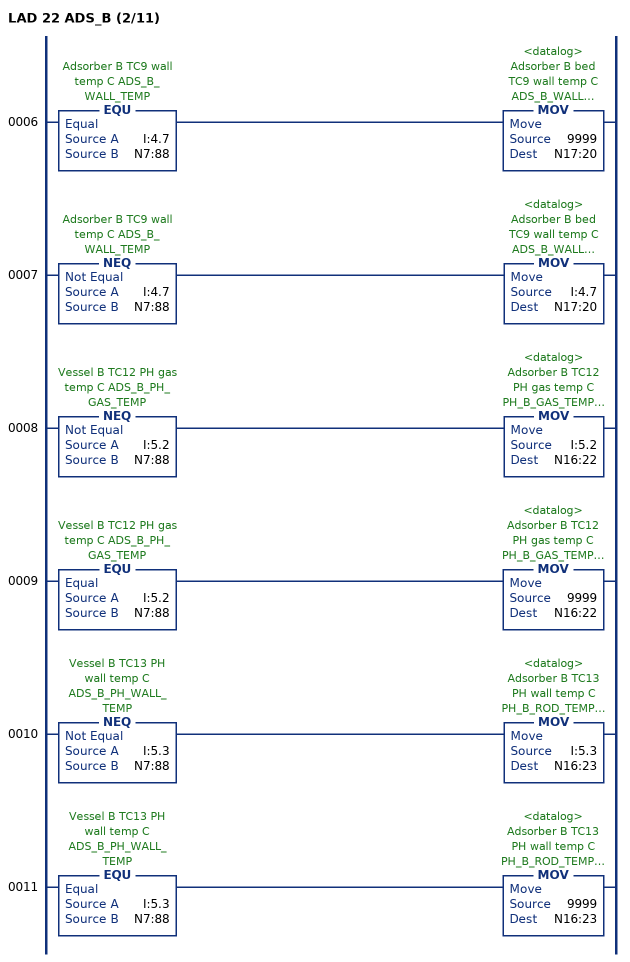
% Rung: 6 %
SOR EQU I:4.7 N7:88 MOV 9999 N17:20 EOR
%   I:4.7  ADS_B_WALL_TEMP  "Adsorber B TC9 wall temp C" %
%   N7:88  TC_OPEN_SP  "CONFIG The value read by an open TC input" %
%   N17:20  ADS_B_WALL_TEMP_READ  "<datalog> Adsorber B bed TC9 wall temp C" %
% Rung: 7 %
SOR NEQ I:4.7 N7:88 MOV I:4.7 N17:20 EOR
%   I:4.7  ADS_B_WALL_TEMP  "Adsorber B TC9 wall temp C" %
%   N7:88  TC_OPEN_SP  "CONFIG The value read by an open TC input" %
%   N17:20  ADS_B_WALL_TEMP_READ  "<datalog> Adsorber B bed TC9 wall temp C" %
% Rung: 8 %
SOR NEQ I:5.2 N7:88 MOV I:5.2 N16:22 EOR
%   I:5.2  ADS_B_PH_GAS_TEMP  "Vessel B TC12 PH gas temp C" %
%   N7:88  TC_OPEN_SP  "CONFIG The value read by an open TC input" %
%   N16:22  PH_B_GAS_TEMP_READ  "<datalog> Adsorber B TC12 PH gas temp C" %
% Rung: 9 %
SOR EQU I:5.2 N7:88 MOV 9999 N16:22 EOR
%   I:5.2  ADS_B_PH_GAS_TEMP  "Vessel B TC12 PH gas temp C" %
%   N7:88  TC_OPEN_SP  "CONFIG The value read by an open TC input" %
%   N16:22  PH_B_GAS_TEMP_READ  "<datalog> Adsorber B TC12 PH gas temp C" %
% Rung: 10 %
SOR NEQ I:5.3 N7:88 MOV I:5.3 N16:23 EOR
%   I:5.3  ADS_B_PH_WALL_TEMP  "Vessel B TC13 PH wall temp C" %
%   N7:88  TC_OPEN_SP  "CONFIG The value read by an open TC input" %
%   N16:23  PH_B_ROD_TEMP_READ  "<datalog> Adsorber B TC13 PH wall temp C" %
% Rung: 11 %
SOR EQU I:5.3 N7:88 MOV 9999 N16:23 EOR
%   I:5.3  ADS_B_PH_WALL_TEMP  "Vessel B TC13 PH wall temp C" %
%   N7:88  TC_OPEN_SP  "CONFIG The value read by an open TC input" %
%   N16:23  PH_B_ROD_TEMP_READ  "<datalog> Adsorber B TC13 PH wall temp C" %

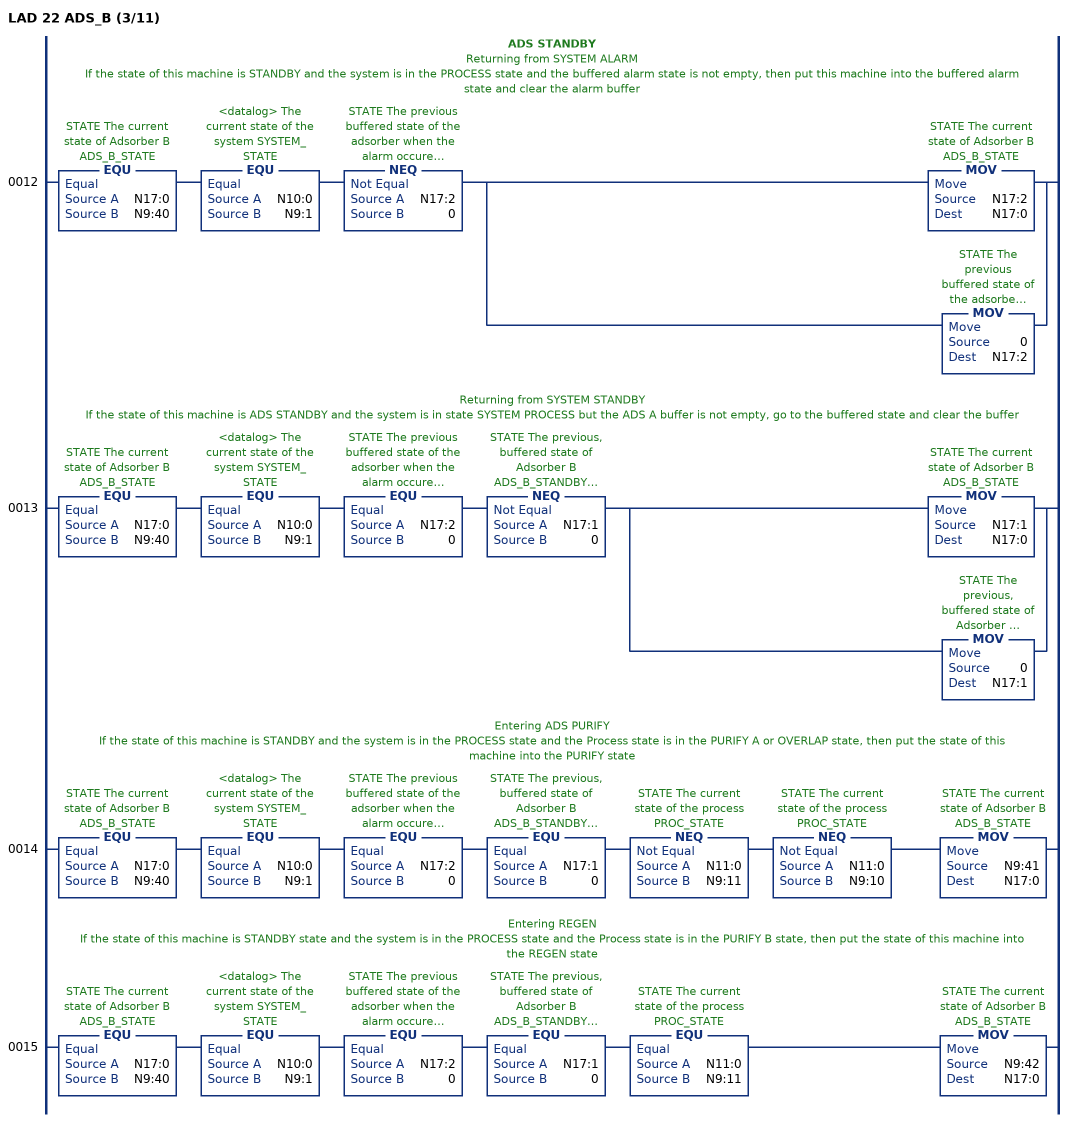
% Rung: 12 %
% TITLE: ADS STANDBY %
% Returning from SYSTEM ALARM
% If the state of this machine is STANDBY and the system is in the PROCESS state and the buffered alarm state is not empty, then put this machine into the buffered alarm state and clear the alarm buffer %
SOR EQU N17:0 N9:40 EQU N10:0 N9:1 NEQ N17:2 0 BST MOV N17:2 N17:0 NXB MOV 0 N17:2 BND EOR
%   N17:0  ADS_B_STATE  "STATE The current state of Adsorber B" %
%   N9:40  ADS_STANDBY  "STATE ADS Standby" %
%   N10:0  SYSTEM_STATE  "<datalog> The current state of the system" %
%   N9:1  SYSTEM_PROCESS  "STATE System Process" %
%   N17:2  ADS_B_SYS_ALARM_BUFR  "STATE The previous buffered state of the adsorber when the alarm occured" %
% Rung: 13 %
% Returning from SYSTEM STANDBY
% If the state of this machine is ADS STANDBY and the system is in state SYSTEM PROCESS but the ADS A buffer is not empty, go to the buffered state and clear the buffer %
SOR EQU N17:0 N9:40 EQU N10:0 N9:1 EQU N17:2 0 NEQ N17:1 0 BST MOV N17:1 N17:0 NXB MOV 0 N17:1 BND EOR
%   N17:0  ADS_B_STATE  "STATE The current state of Adsorber B" %
%   N9:40  ADS_STANDBY  "STATE ADS Standby" %
%   N10:0  SYSTEM_STATE  "<datalog> The current state of the system" %
%   N9:1  SYSTEM_PROCESS  "STATE System Process" %
%   N17:2  ADS_B_SYS_ALARM_BUFR  "STATE The previous buffered state of the adsorber when the alarm occured" %
%   N17:1  ADS_B_STANDBY_BUFFER  "STATE The previous, buffered state of Adsorber B" %
% Rung: 14 %
% Entering ADS PURIFY
% If the state of this machine is STANDBY and the system is in the PROCESS state and the Process state is in the PURIFY A or OVERLAP state, then put the state of this machine into the PURIFY state %
SOR EQU N17:0 N9:40 EQU N10:0 N9:1 EQU N17:2 0 EQU N17:1 0 NEQ N11:0 N9:11 NEQ N11:0 N9:10 MOV N9:41 N17:0 EOR
%   N17:0  ADS_B_STATE  "STATE The current state of Adsorber B" %
%   N9:40  ADS_STANDBY  "STATE ADS Standby" %
%   N10:0  SYSTEM_STATE  "<datalog> The current state of the system" %
%   N9:1  SYSTEM_PROCESS  "STATE System Process" %
%   N17:2  ADS_B_SYS_ALARM_BUFR  "STATE The previous buffered state of the adsorber when the alarm occured" %
%   N17:1  ADS_B_STANDBY_BUFFER  "STATE The previous, buffered state of Adsorber B" %
%   N11:0  PROC_STATE  "STATE The current state of the process" %
%   N9:11  PROC_REGEN_B  "STATE Process Purify A" %
%   N9:10  PROCESS_STANDBY %
%   N9:41  ADS_PURIFY  "STATE ADS Purify" %
% Rung: 15 %
% Entering REGEN
% If the state of this machine is STANDBY state and the system is in the PROCESS state and the Process state is in the PURIFY B state, then put the state of this machine into the REGEN state %
SOR EQU N17:0 N9:40 EQU N10:0 N9:1 EQU N17:2 0 EQU N17:1 0 EQU N11:0 N9:11 MOV N9:42 N17:0 EOR
%   N17:0  ADS_B_STATE  "STATE The current state of Adsorber B" %
%   N9:40  ADS_STANDBY  "STATE ADS Standby" %
%   N10:0  SYSTEM_STATE  "<datalog> The current state of the system" %
%   N9:1  SYSTEM_PROCESS  "STATE System Process" %
%   N17:2  ADS_B_SYS_ALARM_BUFR  "STATE The previous buffered state of the adsorber when the alarm occured" %
%   N17:1  ADS_B_STANDBY_BUFFER  "STATE The previous, buffered state of Adsorber B" %
%   N11:0  PROC_STATE  "STATE The current state of the process" %
%   N9:11  PROC_REGEN_B  "STATE Process Purify A" %
%   N9:42  ADS_REGEN  "STATE ADS Regen" %

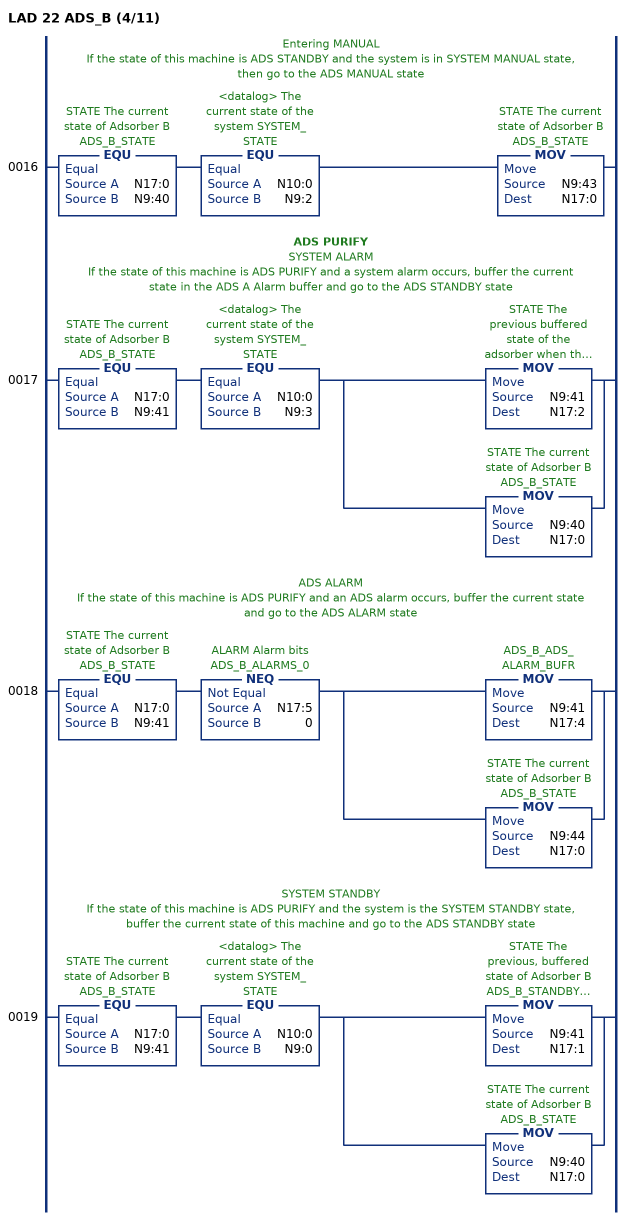
% Rung: 16 %
% Entering MANUAL
% If the state of this machine is ADS STANDBY and the system is in SYSTEM MANUAL state, then go to the ADS MANUAL state %
SOR EQU N17:0 N9:40 EQU N10:0 N9:2 MOV N9:43 N17:0 EOR
%   N17:0  ADS_B_STATE  "STATE The current state of Adsorber B" %
%   N9:40  ADS_STANDBY  "STATE ADS Standby" %
%   N10:0  SYSTEM_STATE  "<datalog> The current state of the system" %
%   N9:2  SYSTEM_MANUAL  "STATE System Manual" %
%   N9:43  ADS_MANUAL  "STATE ADS Manual" %
% Rung: 17 %
% TITLE: ADS PURIFY %
% SYSTEM ALARM
% If the state of this machine is ADS PURIFY and a system alarm occurs, buffer the current state in the ADS A Alarm buffer and go to the ADS STANDBY state %
SOR EQU N17:0 N9:41 EQU N10:0 N9:3 BST MOV N9:41 N17:2 NXB MOV N9:40 N17:0 BND EOR
%   N17:0  ADS_B_STATE  "STATE The current state of Adsorber B" %
%   N9:41  ADS_PURIFY  "STATE ADS Purify" %
%   N10:0  SYSTEM_STATE  "<datalog> The current state of the system" %
%   N9:3  SYSTEM_ALARM  "STATE System Alarm" %
%   N17:2  ADS_B_SYS_ALARM_BUFR  "STATE The previous buffered state of the adsorber when the alarm occured" %
%   N9:40  ADS_STANDBY  "STATE ADS Standby" %
% Rung: 18 %
% ADS ALARM
% If the state of this machine is ADS PURIFY and an ADS alarm occurs, buffer the current state and go to the ADS ALARM state %
SOR EQU N17:0 N9:41 NEQ N17:5 0 BST MOV N9:41 N17:4 NXB MOV N9:44 N17:0 BND EOR
%   N17:0  ADS_B_STATE  "STATE The current state of Adsorber B" %
%   N9:41  ADS_PURIFY  "STATE ADS Purify" %
%   N17:5  ADS_B_ALARMS_0  "ALARM Alarm bits" %
%   N17:4  ADS_B_ADS_ALARM_BUFR %
%   N9:44  ADS_ALARM  "STATE ADS Alarm" %
% Rung: 19 %
% SYSTEM STANDBY
% If the state of this machine is ADS PURIFY and the system is the SYSTEM STANDBY state, buffer the current state of this machine and go to the ADS STANDBY state %
SOR EQU N17:0 N9:41 EQU N10:0 N9:0 BST MOV N9:41 N17:1 NXB MOV N9:40 N17:0 BND EOR
%   N17:0  ADS_B_STATE  "STATE The current state of Adsorber B" %
%   N9:41  ADS_PURIFY  "STATE ADS Purify" %
%   N10:0  SYSTEM_STATE  "<datalog> The current state of the system" %
%   N9:0  SYSTEM_STANDBY  "STATE System Standby" %
%   N17:1  ADS_B_STANDBY_BUFFER  "STATE The previous, buffered state of Adsorber B" %
%   N9:40  ADS_STANDBY  "STATE ADS Standby" %

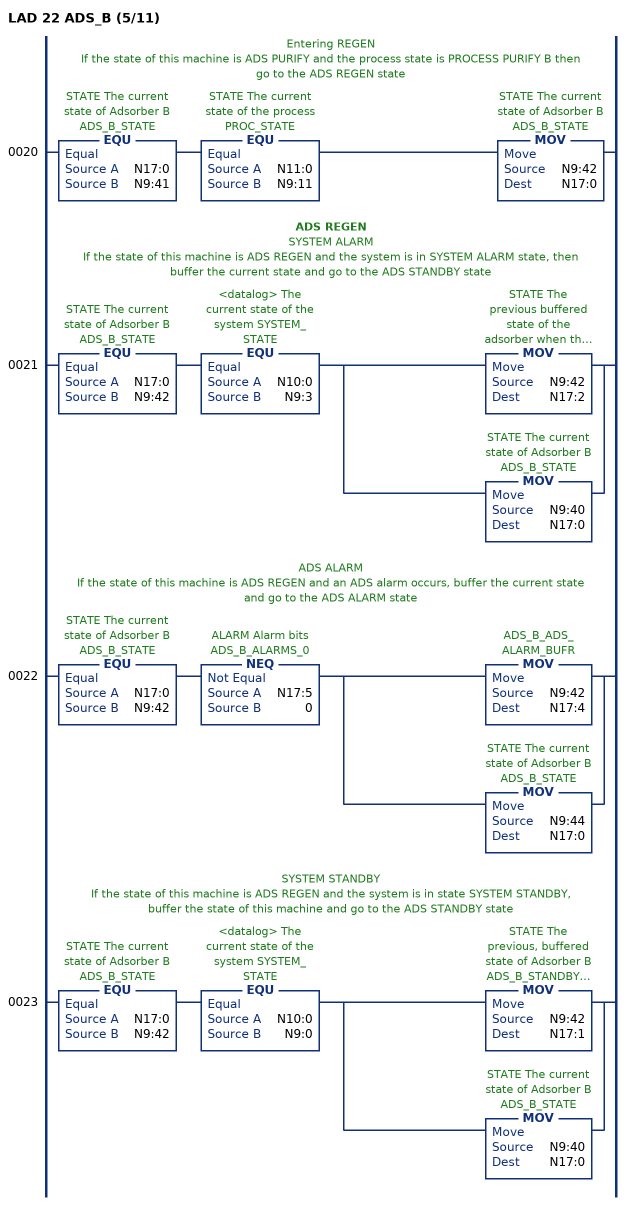
% Rung: 20 %
% Entering REGEN
% If the state of this machine is ADS PURIFY and the process state is PROCESS PURIFY B then go to the ADS REGEN state %
SOR EQU N17:0 N9:41 EQU N11:0 N9:11 MOV N9:42 N17:0 EOR
%   N17:0  ADS_B_STATE  "STATE The current state of Adsorber B" %
%   N9:41  ADS_PURIFY  "STATE ADS Purify" %
%   N11:0  PROC_STATE  "STATE The current state of the process" %
%   N9:11  PROC_REGEN_B  "STATE Process Purify A" %
%   N9:42  ADS_REGEN  "STATE ADS Regen" %
% Rung: 21 %
% TITLE: ADS REGEN %
% SYSTEM ALARM
% If the state of this machine is ADS REGEN and the system is in SYSTEM ALARM state, then buffer the current state and go to the ADS STANDBY state %
SOR EQU N17:0 N9:42 EQU N10:0 N9:3 BST MOV N9:42 N17:2 NXB MOV N9:40 N17:0 BND EOR
%   N17:0  ADS_B_STATE  "STATE The current state of Adsorber B" %
%   N9:42  ADS_REGEN  "STATE ADS Regen" %
%   N10:0  SYSTEM_STATE  "<datalog> The current state of the system" %
%   N9:3  SYSTEM_ALARM  "STATE System Alarm" %
%   N17:2  ADS_B_SYS_ALARM_BUFR  "STATE The previous buffered state of the adsorber when the alarm occured" %
%   N9:40  ADS_STANDBY  "STATE ADS Standby" %
% Rung: 22 %
% ADS ALARM
% If the state of this machine is ADS REGEN and an ADS alarm occurs, buffer the current state and go to the ADS ALARM state %
SOR EQU N17:0 N9:42 NEQ N17:5 0 BST MOV N9:42 N17:4 NXB MOV N9:44 N17:0 BND EOR
%   N17:0  ADS_B_STATE  "STATE The current state of Adsorber B" %
%   N9:42  ADS_REGEN  "STATE ADS Regen" %
%   N17:5  ADS_B_ALARMS_0  "ALARM Alarm bits" %
%   N17:4  ADS_B_ADS_ALARM_BUFR %
%   N9:44  ADS_ALARM  "STATE ADS Alarm" %
% Rung: 23 %
% SYSTEM STANDBY
% If the state of this machine is ADS REGEN and the system is in state SYSTEM STANDBY, buffer the state of this machine and go to the ADS STANDBY state %
SOR EQU N17:0 N9:42 EQU N10:0 N9:0 BST MOV N9:42 N17:1 NXB MOV N9:40 N17:0 BND EOR
%   N17:0  ADS_B_STATE  "STATE The current state of Adsorber B" %
%   N9:42  ADS_REGEN  "STATE ADS Regen" %
%   N10:0  SYSTEM_STATE  "<datalog> The current state of the system" %
%   N9:0  SYSTEM_STANDBY  "STATE System Standby" %
%   N17:1  ADS_B_STANDBY_BUFFER  "STATE The previous, buffered state of Adsorber B" %
%   N9:40  ADS_STANDBY  "STATE ADS Standby" %

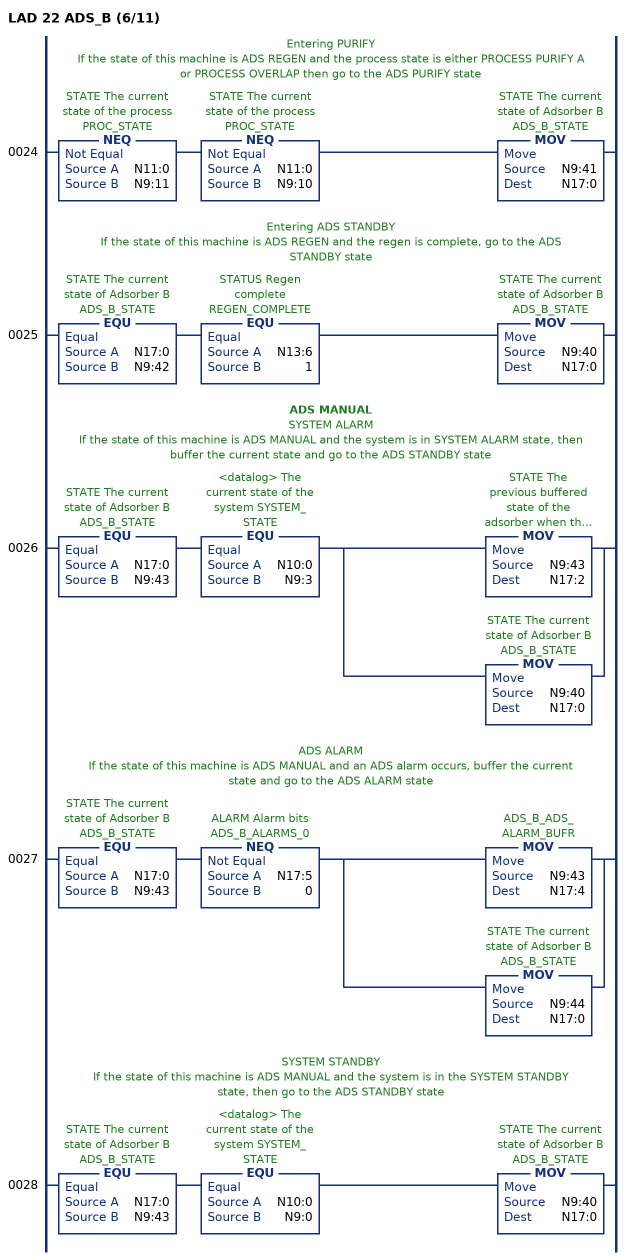
% Rung: 24 %
% Entering PURIFY
% If the state of this machine is ADS REGEN and the process state is either PROCESS PURIFY A or PROCESS OVERLAP then go to the ADS PURIFY state %
SOR NEQ N11:0 N9:11 NEQ N11:0 N9:10 MOV N9:41 N17:0 EOR
%   N11:0  PROC_STATE  "STATE The current state of the process" %
%   N9:11  PROC_REGEN_B  "STATE Process Purify A" %
%   N9:10  PROCESS_STANDBY %
%   N9:41  ADS_PURIFY  "STATE ADS Purify" %
%   N17:0  ADS_B_STATE  "STATE The current state of Adsorber B" %
% Rung: 25 %
% Entering ADS STANDBY
% If the state of this machine is ADS REGEN and the regen is complete, go to the ADS STANDBY state %
SOR EQU N17:0 N9:42 EQU N13:6 1 MOV N9:40 N17:0 EOR
%   N17:0  ADS_B_STATE  "STATE The current state of Adsorber B" %
%   N9:42  ADS_REGEN  "STATE ADS Regen" %
%   N13:6  REGEN_COMPLETE  "STATUS Regen complete" %
%   N9:40  ADS_STANDBY  "STATE ADS Standby" %
% Rung: 26 %
% TITLE: ADS MANUAL %
% SYSTEM ALARM
% If the state of this machine is ADS MANUAL and the system is in SYSTEM ALARM state, then buffer the current state and go to the ADS STANDBY state %
SOR EQU N17:0 N9:43 EQU N10:0 N9:3 BST MOV N9:43 N17:2 NXB MOV N9:40 N17:0 BND EOR
%   N17:0  ADS_B_STATE  "STATE The current state of Adsorber B" %
%   N9:43  ADS_MANUAL  "STATE ADS Manual" %
%   N10:0  SYSTEM_STATE  "<datalog> The current state of the system" %
%   N9:3  SYSTEM_ALARM  "STATE System Alarm" %
%   N17:2  ADS_B_SYS_ALARM_BUFR  "STATE The previous buffered state of the adsorber when the alarm occured" %
%   N9:40  ADS_STANDBY  "STATE ADS Standby" %
% Rung: 27 %
% ADS ALARM
% If the state of this machine is ADS MANUAL and an ADS alarm occurs, buffer the current state and go to the ADS ALARM state %
SOR EQU N17:0 N9:43 NEQ N17:5 0 BST MOV N9:43 N17:4 NXB MOV N9:44 N17:0 BND EOR
%   N17:0  ADS_B_STATE  "STATE The current state of Adsorber B" %
%   N9:43  ADS_MANUAL  "STATE ADS Manual" %
%   N17:5  ADS_B_ALARMS_0  "ALARM Alarm bits" %
%   N17:4  ADS_B_ADS_ALARM_BUFR %
%   N9:44  ADS_ALARM  "STATE ADS Alarm" %
% Rung: 28 %
% SYSTEM STANDBY
% If the state of this machine is ADS MANUAL and the system is in the SYSTEM STANDBY state, then go to the ADS STANDBY state %
SOR EQU N17:0 N9:43 EQU N10:0 N9:0 MOV N9:40 N17:0 EOR
%   N17:0  ADS_B_STATE  "STATE The current state of Adsorber B" %
%   N9:43  ADS_MANUAL  "STATE ADS Manual" %
%   N10:0  SYSTEM_STATE  "<datalog> The current state of the system" %
%   N9:0  SYSTEM_STANDBY  "STATE System Standby" %
%   N9:40  ADS_STANDBY  "STATE ADS Standby" %

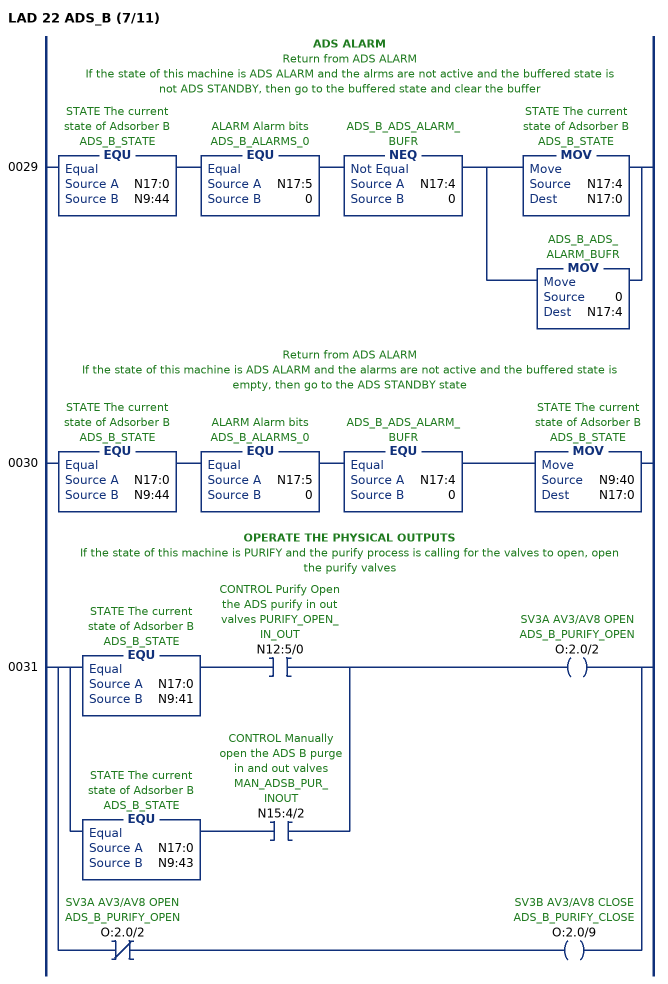
% Rung: 29 %
% TITLE: ADS ALARM %
% Return from ADS ALARM
% If the state of this machine is ADS ALARM and the alrms are not active and the buffered state is not ADS STANDBY, then go to the buffered state and clear the buffer %
SOR EQU N17:0 N9:44 EQU N17:5 0 NEQ N17:4 0 BST MOV N17:4 N17:0 NXB MOV 0 N17:4 BND EOR
%   N17:0  ADS_B_STATE  "STATE The current state of Adsorber B" %
%   N9:44  ADS_ALARM  "STATE ADS Alarm" %
%   N17:5  ADS_B_ALARMS_0  "ALARM Alarm bits" %
%   N17:4  ADS_B_ADS_ALARM_BUFR %
% Rung: 30 %
% Return from ADS ALARM
% If the state of this machine is ADS ALARM and the alarms are not active and the buffered state is empty, then go to the ADS STANDBY state %
SOR EQU N17:0 N9:44 EQU N17:5 0 EQU N17:4 0 MOV N9:40 N17:0 EOR
%   N17:0  ADS_B_STATE  "STATE The current state of Adsorber B" %
%   N9:44  ADS_ALARM  "STATE ADS Alarm" %
%   N17:5  ADS_B_ALARMS_0  "ALARM Alarm bits" %
%   N17:4  ADS_B_ADS_ALARM_BUFR %
%   N9:40  ADS_STANDBY  "STATE ADS Standby" %
% Rung: 31 %
% TITLE: OPERATE THE PHYSICAL OUTPUTS %
% If the state of this machine is PURIFY and the purify process is calling for the valves to open, open the purify valves %
SOR BST BST EQU N17:0 N9:41 XIC N12:5/0 NXB EQU N17:0 N9:43 XIC N15:4/2 BND OTE O:2.0/2 NXB XIO O:2.0/2 OTE O:2.0/9 BND EOR
%   N17:0  ADS_B_STATE  "STATE The current state of Adsorber B" %
%   N9:41  ADS_PURIFY  "STATE ADS Purify" %
%   N12:5/0  PURIFY_OPEN_IN_OUT  "CONTROL Purify Open the ADS purify in out valves" %
%   N9:43  ADS_MANUAL  "STATE ADS Manual" %
%   N15:4/2  MAN_ADSB_PUR_INOUT  "CONTROL Manually open the ADS B purge in and out valves" %
%   O:2.0/2  ADS_B_PURIFY_OPEN  "SV3A AV3/AV8 OPEN" %
%   O:2.0/9  ADS_B_PURIFY_CLOSE  "SV3B AV3/AV8 CLOSE" %

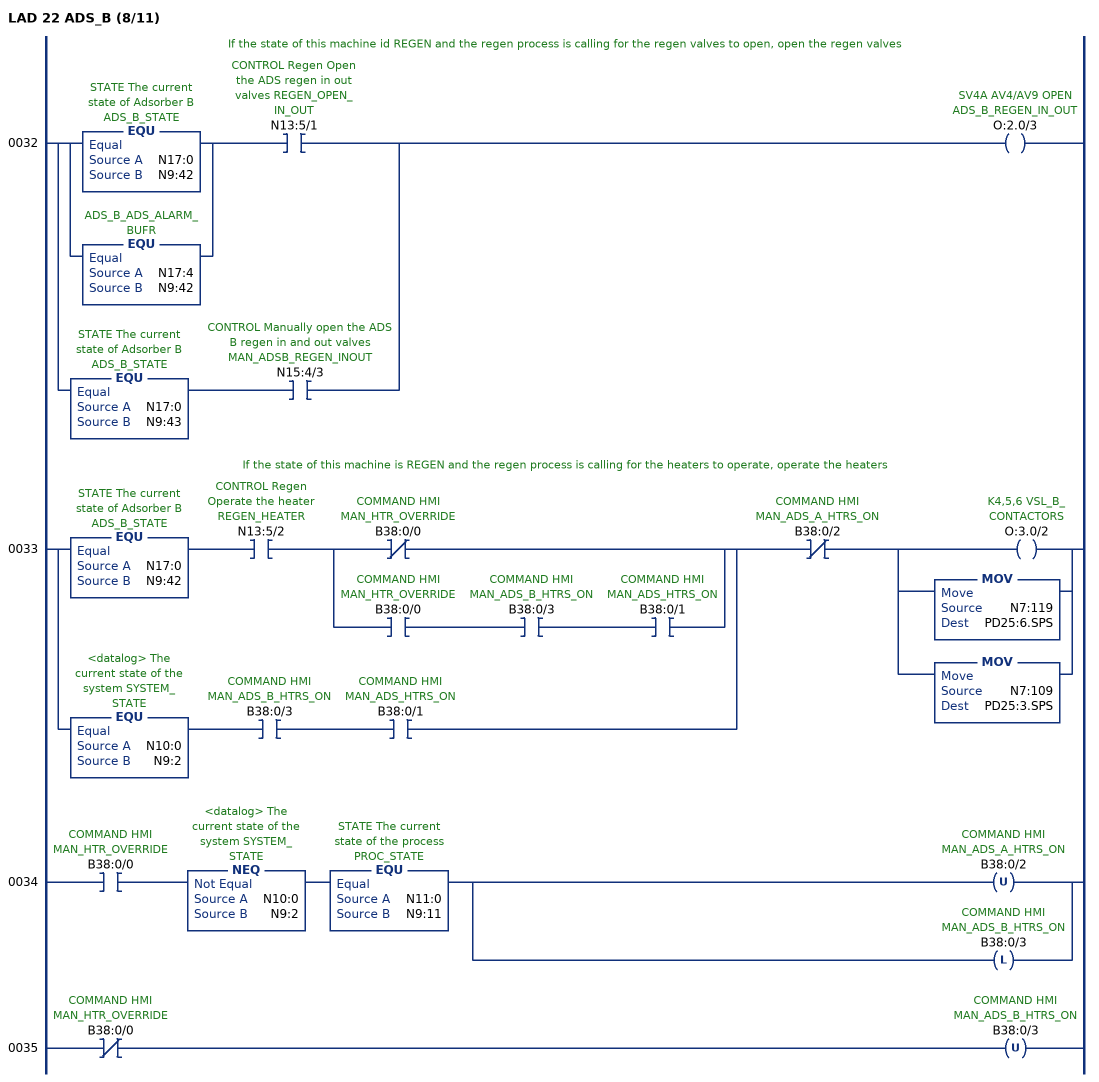
% Rung: 32 %
% If the state of this machine id REGEN and the regen process is calling for the regen valves to open, open the regen valves %
SOR BST BST EQU N17:0 N9:42 NXB EQU N17:4 N9:42 BND XIC N13:5/1 NXB EQU N17:0 N9:43 XIC N15:4/3 BND OTE O:2.0/3 EOR
%   N17:0  ADS_B_STATE  "STATE The current state of Adsorber B" %
%   N9:42  ADS_REGEN  "STATE ADS Regen" %
%   N17:4  ADS_B_ADS_ALARM_BUFR %
%   N13:5/1  REGEN_OPEN_IN_OUT  "CONTROL Regen Open the ADS regen in out valves" %
%   N9:43  ADS_MANUAL  "STATE ADS Manual" %
%   N15:4/3  MAN_ADSB_REGEN_INOUT  "CONTROL Manually open the ADS B regen in and out valves" %
%   O:2.0/3  ADS_B_REGEN_IN_OUT  "SV4A AV4/AV9 OPEN" %
% Rung: 33 %
% If the state of this machine is REGEN and the regen process is calling for the heaters to operate, operate the heaters %
SOR BST EQU N17:0 N9:42 XIC N13:5/2 BST XIO B38:0/0 NXB XIC B38:0/0 XIC B38:0/3 XIC B38:0/1 BND NXB EQU N10:0 N9:2 XIC B38:0/3 XIC B38:0/1 BND XIO B38:0/2 BST OTE O:3.0/2 NXB MOV N7:119 PD25:6.SPS NXB MOV N7:109 PD25:3.SPS BND EOR
%   N17:0  ADS_B_STATE  "STATE The current state of Adsorber B" %
%   N9:42  ADS_REGEN  "STATE ADS Regen" %
%   N13:5/2  REGEN_HEATER  "CONTROL Regen Operate the heater" %
%   B38:0/0  MAN_HTR_OVERRIDE  "COMMAND HMI" %
%   B38:0/3  MAN_ADS_B_HTRS_ON  "COMMAND HMI" %
%   B38:0/1  MAN_ADS_HTRS_ON  "COMMAND HMI" %
%   N10:0  SYSTEM_STATE  "<datalog> The current state of the system" %
%   N9:2  SYSTEM_MANUAL  "STATE System Manual" %
%   B38:0/2  MAN_ADS_A_HTRS_ON  "COMMAND HMI" %
%   O:3.0/2  VSL_B_CONTACTORS  "K4,5,6" %
%   N7:119  PREHEATER_SP  "<datalog> CONTROL Preheater PID Setpoint" %
%   N7:109  BLANKET_SP  "CONTROL Blanket PID Setpoint" %
% Rung: 34 %
SOR XIC B38:0/0 NEQ N10:0 N9:2 EQU N11:0 N9:11 BST OTU B38:0/2 NXB OTL B38:0/3 BND EOR
%   B38:0/0  MAN_HTR_OVERRIDE  "COMMAND HMI" %
%   N10:0  SYSTEM_STATE  "<datalog> The current state of the system" %
%   N9:2  SYSTEM_MANUAL  "STATE System Manual" %
%   N11:0  PROC_STATE  "STATE The current state of the process" %
%   N9:11  PROC_REGEN_B  "STATE Process Purify A" %
%   B38:0/2  MAN_ADS_A_HTRS_ON  "COMMAND HMI" %
%   B38:0/3  MAN_ADS_B_HTRS_ON  "COMMAND HMI" %
% Rung: 35 %
SOR XIO B38:0/0 OTU B38:0/3 EOR
%   B38:0/0  MAN_HTR_OVERRIDE  "COMMAND HMI" %
%   B38:0/3  MAN_ADS_B_HTRS_ON  "COMMAND HMI" %

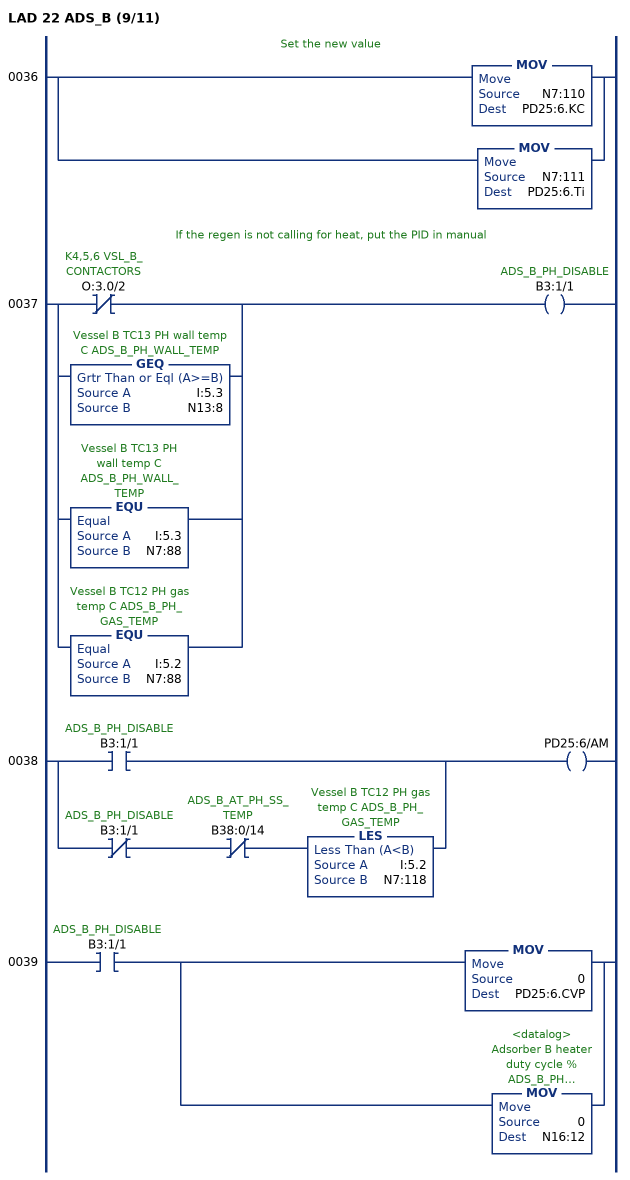
% Rung: 36 %
% Set the new value %
SOR BST MOV N7:110 PD25:6.KC NXB MOV N7:111 PD25:6.Ti BND EOR
%   N7:110  PREHEATER_P  "<datalog> CONFIG Preheater Proportional Gain New" %
%   N7:111  PREHEATER_I  "<datalog> CONFIG Preheater Integral Gain New" %
% Rung: 37 %
% If the regen is not calling for heat, put the PID in manual %
SOR BST XIO O:3.0/2 NXB GEQ I:5.3 N13:8 NXB EQU I:5.3 N7:88 NXB EQU I:5.2 N7:88 BND OTE B3:1/1 EOR
%   O:3.0/2  VSL_B_CONTACTORS  "K4,5,6" %
%   I:5.3  ADS_B_PH_WALL_TEMP  "Vessel B TC13 PH wall temp C" %
%   N13:8  PH_ROD_LIMIT %
%   N7:88  TC_OPEN_SP  "CONFIG The value read by an open TC input" %
%   I:5.2  ADS_B_PH_GAS_TEMP  "Vessel B TC12 PH gas temp C" %
%   B3:1/1  ADS_B_PH_DISABLE %
% Rung: 38 %
SOR BST XIC B3:1/1 NXB XIO B3:1/1 XIO B38:0/14 LES I:5.2 N7:118 BND OTE PD25:6/AM EOR
%   B3:1/1  ADS_B_PH_DISABLE %
%   B38:0/14  ADS_B_AT_PH_SS_TEMP %
%   I:5.2  ADS_B_PH_GAS_TEMP  "Vessel B TC12 PH gas temp C" %
%   N7:118  PH_SS_TEMP_SP %
% Rung: 39 %
SOR XIC B3:1/1 BST MOV 0 PD25:6.CVP NXB MOV 0 N16:12 BND EOR
%   B3:1/1  ADS_B_PH_DISABLE %
%   N16:12  ADS_B_PH_OUTPUT  "<datalog> Adsorber B heater duty cycle %" %

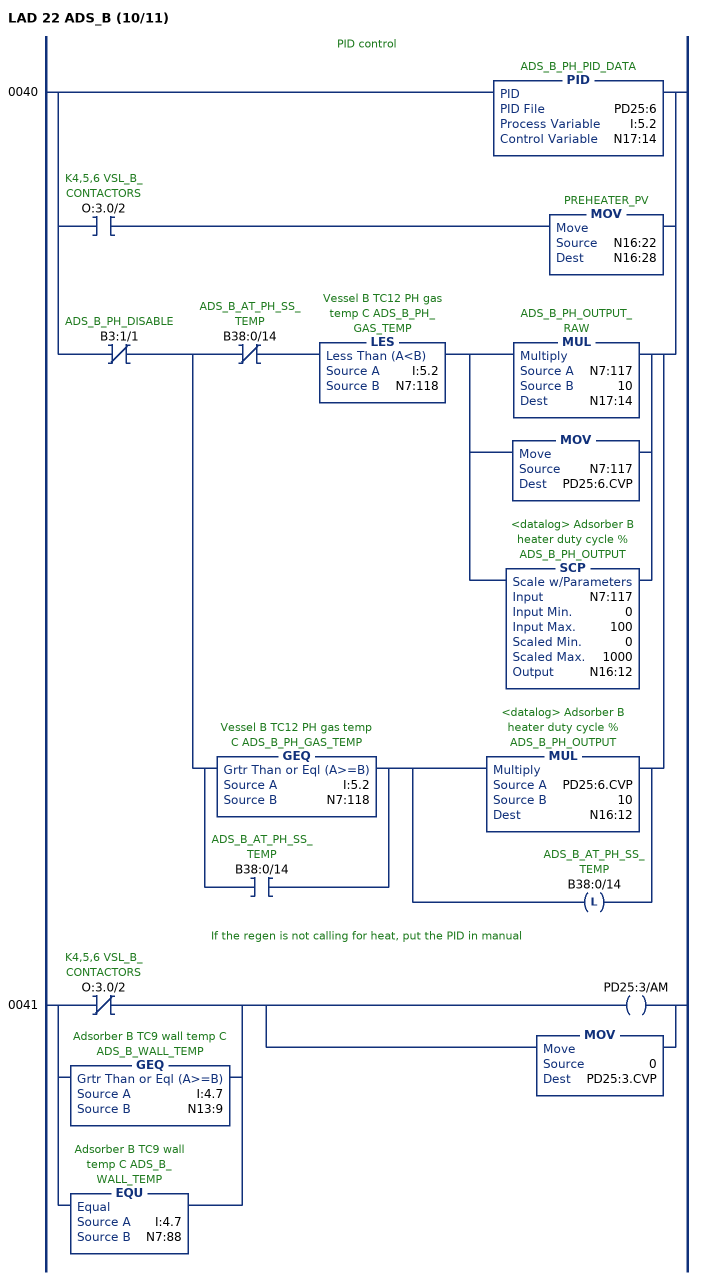
% Rung: 40 %
% PID control %
SOR BST PID PD25:6 I:5.2 N17:14 NXB XIC O:3.0/2 MOV N16:22 N16:28 NXB XIO B3:1/1 BST XIO B38:0/14 LES I:5.2 N7:118 BST MUL N7:117 10 N17:14 NXB MOV N7:117 PD25:6.CVP NXB SCP N7:117 0 100 0 1000 N16:12 BND NXB BST GEQ I:5.2 N7:118 NXB XIC B38:0/14 BND BST MUL PD25:6.CVP 10 N16:12 NXB OTL B38:0/14 BND BND BND EOR
%   PD25:6  ADS_B_PH_PID_DATA %
%   I:5.2  ADS_B_PH_GAS_TEMP  "Vessel B TC12 PH gas temp C" %
%   N17:14  ADS_B_PH_OUTPUT_RAW %
%   O:3.0/2  VSL_B_CONTACTORS  "K4,5,6" %
%   N16:22  PH_B_GAS_TEMP_READ  "<datalog> Adsorber B TC12 PH gas temp C" %
%   N16:28  PREHEATER_PV %
%   B3:1/1  ADS_B_PH_DISABLE %
%   B38:0/14  ADS_B_AT_PH_SS_TEMP %
%   N7:118  PH_SS_TEMP_SP %
%   N7:117  PH_SS_OUTPUT %
%   N16:12  ADS_B_PH_OUTPUT  "<datalog> Adsorber B heater duty cycle %" %
% Rung: 41 %
% If the regen is not calling for heat, put the PID in manual %
SOR BST XIO O:3.0/2 NXB GEQ I:4.7 N13:9 NXB EQU I:4.7 N7:88 BND BST OTE PD25:3/AM NXB MOV 0 PD25:3.CVP BND EOR
%   O:3.0/2  VSL_B_CONTACTORS  "K4,5,6" %
%   I:4.7  ADS_B_WALL_TEMP  "Adsorber B TC9 wall temp C" %
%   N13:9  BLANKET_LIMIT %
%   N7:88  TC_OPEN_SP  "CONFIG The value read by an open TC input" %

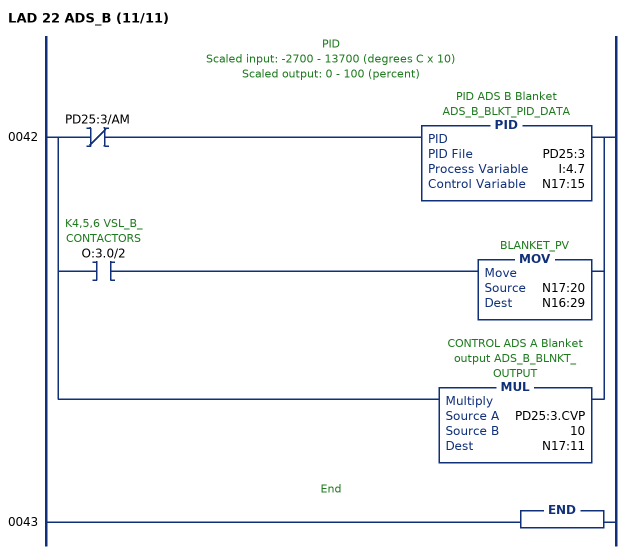
% Rung: 42 %
% PID
% Scaled input: -2700 - 13700 (degrees C x 10)
% Scaled output: 0 - 100 (percent) %
SOR BST XIO PD25:3/AM PID PD25:3 I:4.7 N17:15 NXB XIC O:3.0/2 MOV N17:20 N16:29 NXB MUL PD25:3.CVP 10 N17:11 BND EOR
%   PD25:3  ADS_B_BLKT_PID_DATA  "PID ADS B Blanket" %
%   I:4.7  ADS_B_WALL_TEMP  "Adsorber B TC9 wall temp C" %
%   N17:15  ADS_B_BLKT_OUTPT_RAW  "CONTROL ADS B Blanket PID Output Raw" %
%   O:3.0/2  VSL_B_CONTACTORS  "K4,5,6" %
%   N17:20  ADS_B_WALL_TEMP_READ  "<datalog> Adsorber B bed TC9 wall temp C" %
%   N16:29  BLANKET_PV %
%   N17:11  ADS_B_BLNKT_OUTPUT  "CONTROL ADS A Blanket output" %
% Rung: 43 %
% End %
SOR END EOR

LADDER 23 "ADS_B_FLT"    % Controls the Adsorber B faults %
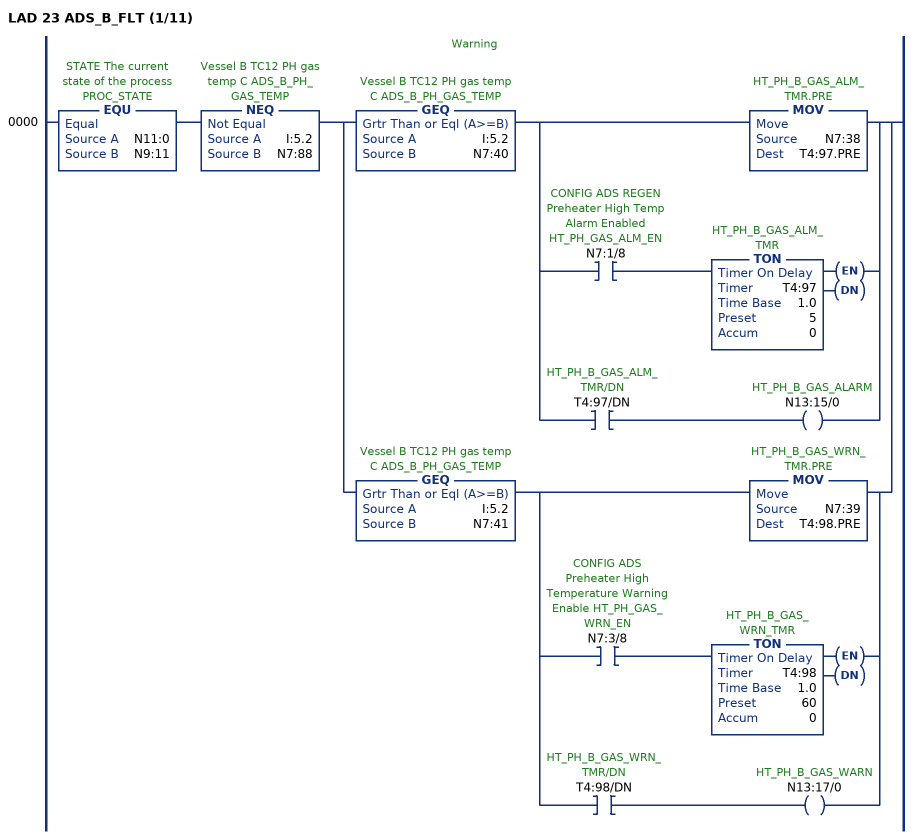
% Rung: 0 %
% Warning %
SOR EQU N11:0 N9:11 NEQ I:5.2 N7:88 BST GEQ I:5.2 N7:40 BST MOV N7:38 T4:97.PRE NXB XIC N7:1/8 TON T4:97 1.0 5 0 NXB XIC T4:97/DN OTE N13:15/0 BND NXB GEQ I:5.2 N7:41 BST MOV N7:39 T4:98.PRE NXB XIC N7:3/8 TON T4:98 1.0 60 0 NXB XIC T4:98/DN OTE N13:17/0 BND BND EOR
%   N11:0  PROC_STATE  "STATE The current state of the process" %
%   N9:11  PROC_REGEN_B  "STATE Process Purify A" %
%   I:5.2  ADS_B_PH_GAS_TEMP  "Vessel B TC12 PH gas temp C" %
%   N7:88  TC_OPEN_SP  "CONFIG The value read by an open TC input" %
%   N7:40  HT_PH_GAS_ALM_SP  "CONFIG ADS Preheater High Temperature Alarm Temperature" %
%   N7:38  HT_PH_GAS_ALM_DLY  "CONFIG ADS Preheater High Temperature Alarm Delay" %
%   T4:97  HT_PH_B_GAS_ALM_TMR %
%   N7:1/8  HT_PH_GAS_ALM_EN  "CONFIG ADS REGEN Preheater High Temp Alarm Enabled" %
%   N13:15/0  HT_PH_B_GAS_ALARM %
%   N7:41  HT_PH_GAS_WRN_SP  "CONFIG ADS Preheater High Temperature Warning Temperature" %
%   N7:39  HT_PH_GAS_WRN_DLY  "CONFIG ADS Preheater High Temperature Warning Delay" %
%   T4:98  HT_PH_B_GAS_WRN_TMR %
%   N7:3/8  HT_PH_GAS_WRN_EN  "CONFIG ADS Preheater High Temperature Warning Enable" %
%   N13:17/0  HT_PH_B_GAS_WARN %

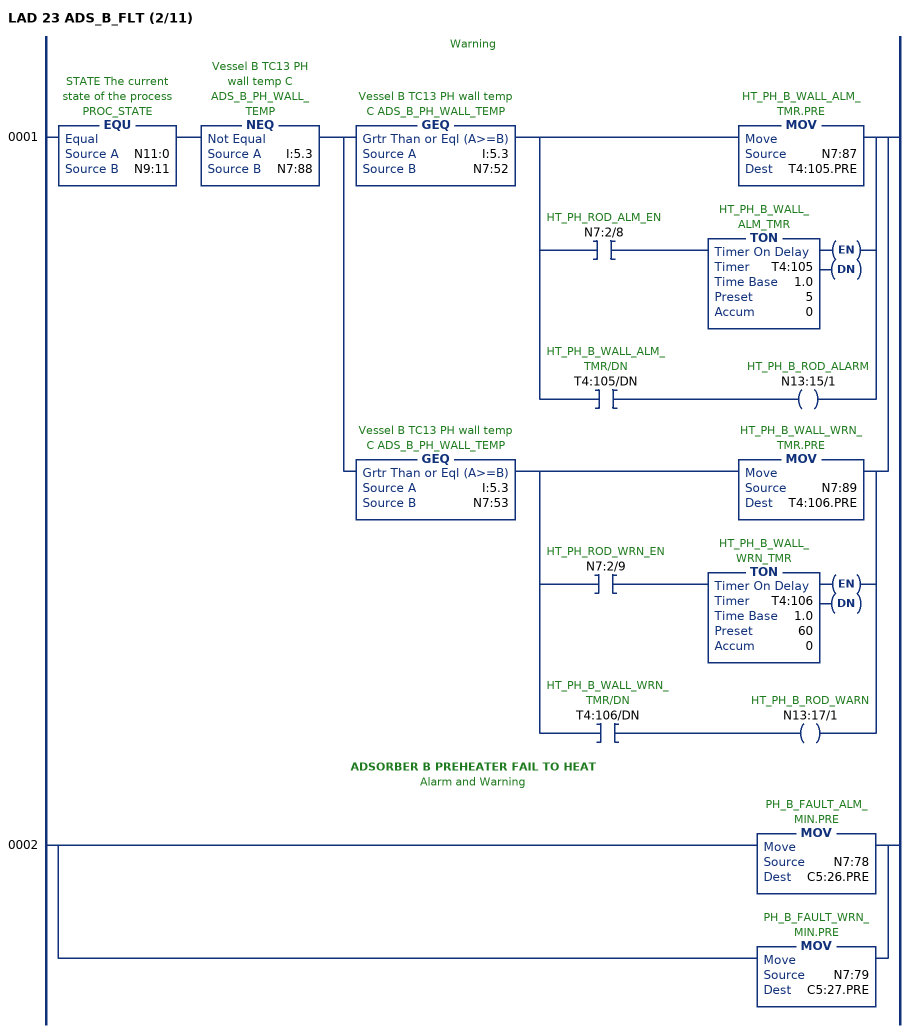
% Rung: 1 %
% Warning %
SOR EQU N11:0 N9:11 NEQ I:5.3 N7:88 BST GEQ I:5.3 N7:52 BST MOV N7:87 T4:105.PRE NXB XIC N7:2/8 TON T4:105 1.0 5 0 NXB XIC T4:105/DN OTE N13:15/1 BND NXB GEQ I:5.3 N7:53 BST MOV N7:89 T4:106.PRE NXB XIC N7:2/9 TON T4:106 1.0 60 0 NXB XIC T4:106/DN OTE N13:17/1 BND BND EOR
%   N11:0  PROC_STATE  "STATE The current state of the process" %
%   N9:11  PROC_REGEN_B  "STATE Process Purify A" %
%   I:5.3  ADS_B_PH_WALL_TEMP  "Vessel B TC13 PH wall temp C" %
%   N7:88  TC_OPEN_SP  "CONFIG The value read by an open TC input" %
%   N7:52  HT_PH_ROD_ALM_SP %
%   N7:87  HT_PH_ROD_ALM_DLY %
%   T4:105  HT_PH_B_WALL_ALM_TMR %
%   N7:2/8  HT_PH_ROD_ALM_EN %
%   N13:15/1  HT_PH_B_ROD_ALARM %
%   N7:53  HT_PH_ROD_WRN_SP %
%   N7:89  HT_PH_ROD_WRN_DLY %
%   T4:106  HT_PH_B_WALL_WRN_TMR %
%   N7:2/9  HT_PH_ROD_WRN_EN %
%   N13:17/1  HT_PH_B_ROD_WARN %
% Rung: 2 %
% TITLE: ADSORBER B PREHEATER FAIL TO HEAT %
% Alarm and Warning %
SOR BST MOV N7:78 C5:26.PRE NXB MOV N7:79 C5:27.PRE BND EOR
%   N7:78  PH_FAULT_ALM_DLY %
%   C5:26  PH_B_FAULT_ALM_MIN %
%   N7:79  PH_FAULT_WRN_DLY %
%   C5:27  PH_B_FAULT_WRN_MIN %

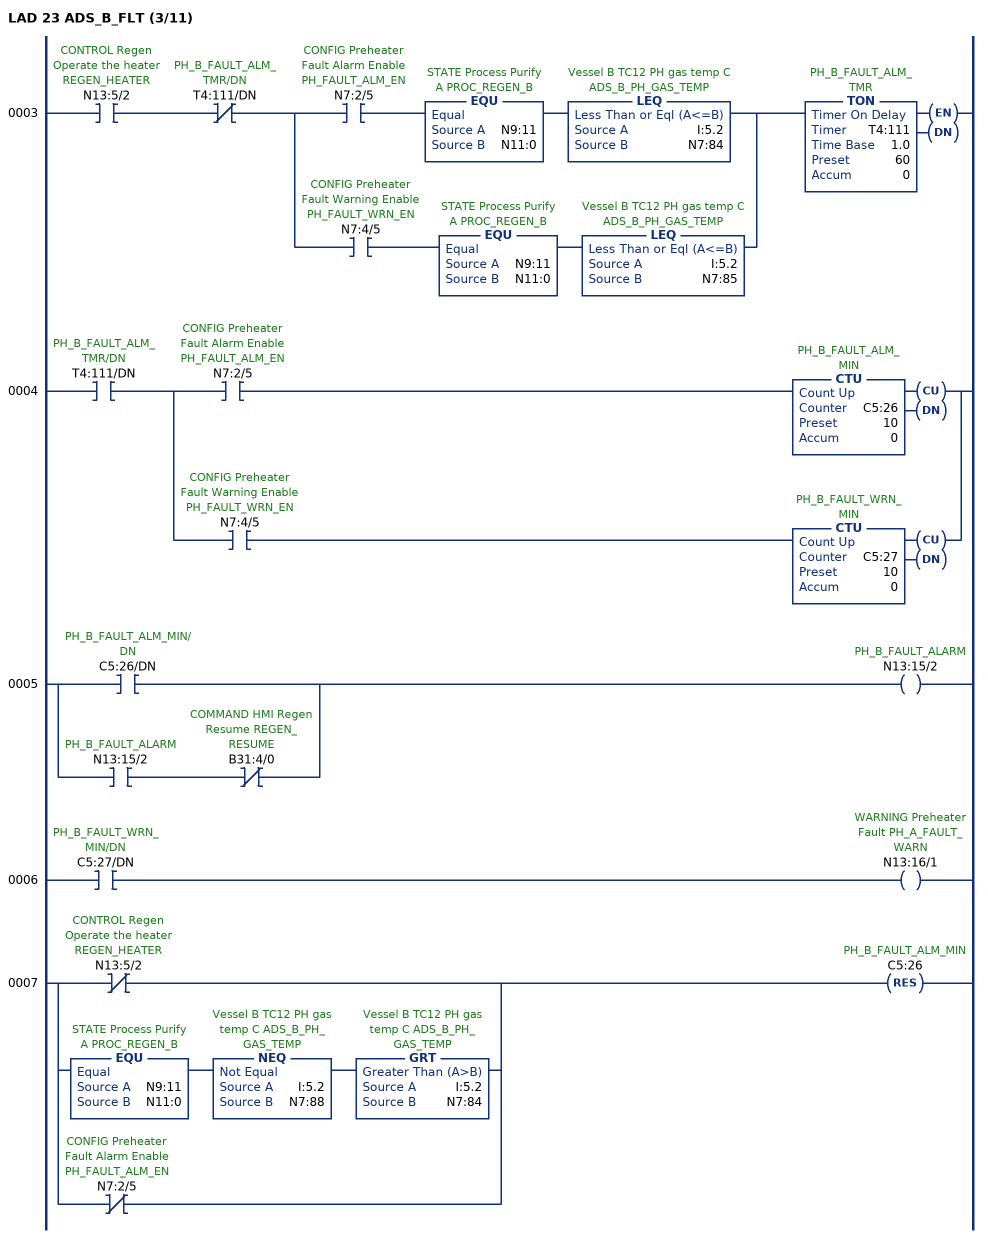
% Rung: 3 %
SOR XIC N13:5/2 XIO T4:111/DN BST XIC N7:2/5 EQU N9:11 N11:0 LEQ I:5.2 N7:84 NXB XIC N7:4/5 EQU N9:11 N11:0 LEQ I:5.2 N7:85 BND TON T4:111 1.0 60 0 EOR
%   N13:5/2  REGEN_HEATER  "CONTROL Regen Operate the heater" %
%   T4:111  PH_B_FAULT_ALM_TMR %
%   N7:2/5  PH_FAULT_ALM_EN  "CONFIG Preheater Fault Alarm Enable" %
%   N9:11  PROC_REGEN_B  "STATE Process Purify A" %
%   N11:0  PROC_STATE  "STATE The current state of the process" %
%   I:5.2  ADS_B_PH_GAS_TEMP  "Vessel B TC12 PH gas temp C" %
%   N7:84  PH_FAULT_ALARM_SP  "CONFIG Preheater Temperature Delta Alarm Setpoint" %
%   N7:4/5  PH_FAULT_WRN_EN  "CONFIG Preheater Fault Warning Enable" %
%   N7:85  PH_FAULT_WARN_SP %
% Rung: 4 %
SOR XIC T4:111/DN BST XIC N7:2/5 CTU C5:26 10 0 NXB XIC N7:4/5 CTU C5:27 10 0 BND EOR
%   T4:111  PH_B_FAULT_ALM_TMR %
%   N7:2/5  PH_FAULT_ALM_EN  "CONFIG Preheater Fault Alarm Enable" %
%   C5:26  PH_B_FAULT_ALM_MIN %
%   N7:4/5  PH_FAULT_WRN_EN  "CONFIG Preheater Fault Warning Enable" %
%   C5:27  PH_B_FAULT_WRN_MIN %
% Rung: 5 %
SOR BST XIC C5:26/DN NXB XIC N13:15/2 XIO B31:4/0 BND OTE N13:15/2 EOR
%   C5:26  PH_B_FAULT_ALM_MIN %
%   N13:15/2  PH_B_FAULT_ALARM %
%   B31:4/0  REGEN_RESUME  "COMMAND HMI Regen Resume" %
% Rung: 6 %
SOR XIC C5:27/DN OTE N13:16/1 EOR
%   C5:27  PH_B_FAULT_WRN_MIN %
%   N13:16/1  PH_A_FAULT_WARN  "WARNING Preheater Fault" %
% Rung: 7 %
SOR BST XIO N13:5/2 NXB EQU N9:11 N11:0 NEQ I:5.2 N7:88 GRT I:5.2 N7:84 NXB XIO N7:2/5 BND RES C5:26 EOR
%   N13:5/2  REGEN_HEATER  "CONTROL Regen Operate the heater" %
%   N9:11  PROC_REGEN_B  "STATE Process Purify A" %
%   N11:0  PROC_STATE  "STATE The current state of the process" %
%   I:5.2  ADS_B_PH_GAS_TEMP  "Vessel B TC12 PH gas temp C" %
%   N7:88  TC_OPEN_SP  "CONFIG The value read by an open TC input" %
%   N7:84  PH_FAULT_ALARM_SP  "CONFIG Preheater Temperature Delta Alarm Setpoint" %
%   N7:2/5  PH_FAULT_ALM_EN  "CONFIG Preheater Fault Alarm Enable" %
%   C5:26  PH_B_FAULT_ALM_MIN %

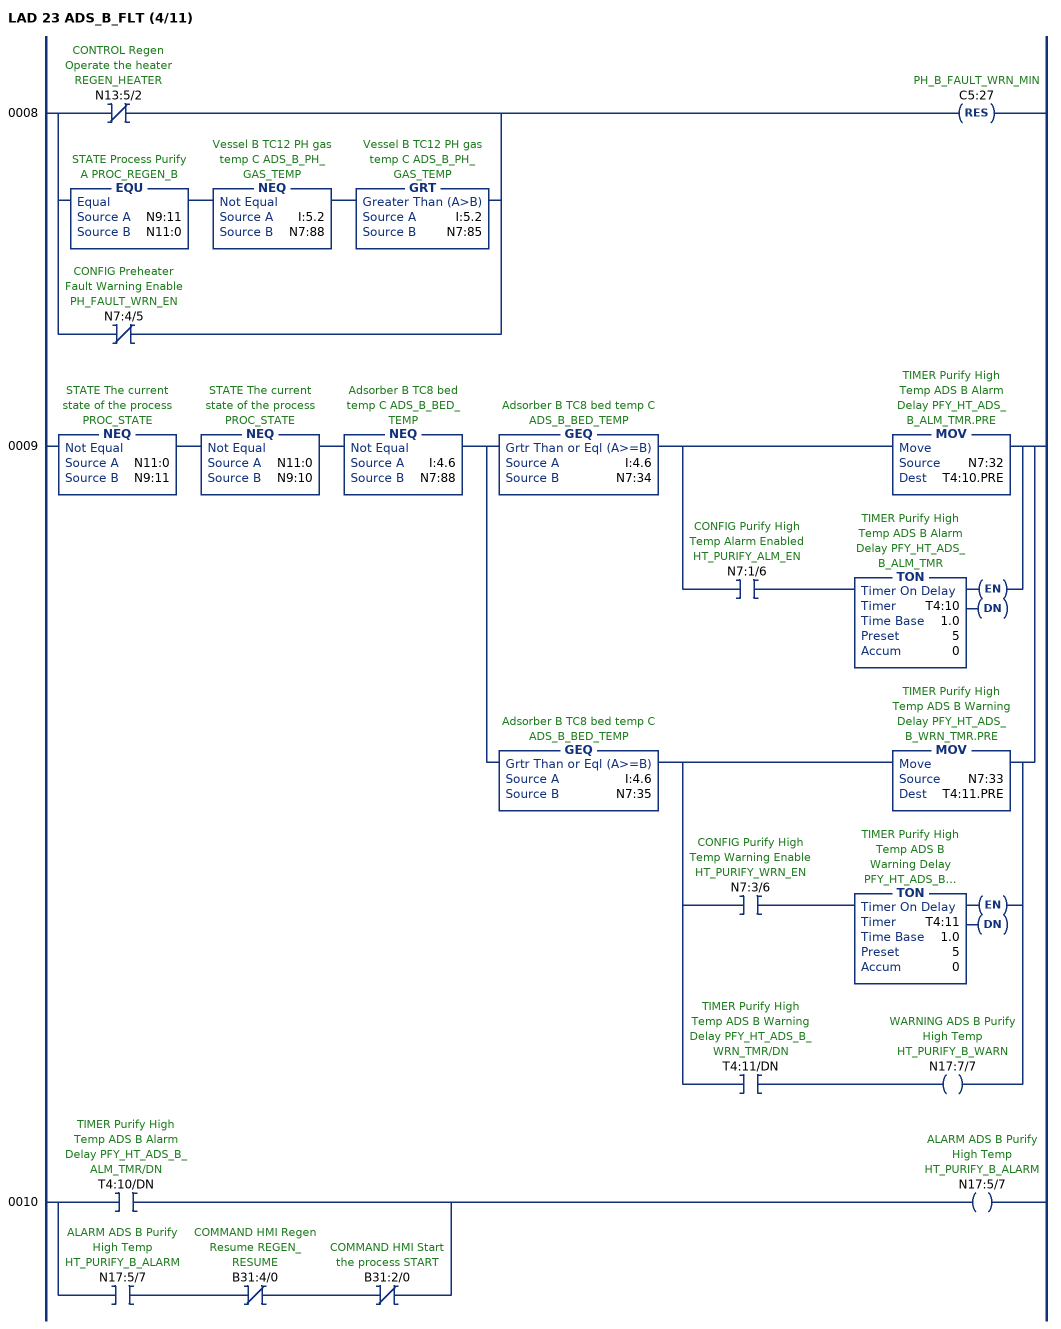
% Rung: 8 %
SOR BST XIO N13:5/2 NXB EQU N9:11 N11:0 NEQ I:5.2 N7:88 GRT I:5.2 N7:85 NXB XIO N7:4/5 BND RES C5:27 EOR
%   N13:5/2  REGEN_HEATER  "CONTROL Regen Operate the heater" %
%   N9:11  PROC_REGEN_B  "STATE Process Purify A" %
%   N11:0  PROC_STATE  "STATE The current state of the process" %
%   I:5.2  ADS_B_PH_GAS_TEMP  "Vessel B TC12 PH gas temp C" %
%   N7:88  TC_OPEN_SP  "CONFIG The value read by an open TC input" %
%   N7:85  PH_FAULT_WARN_SP %
%   N7:4/5  PH_FAULT_WRN_EN  "CONFIG Preheater Fault Warning Enable" %
%   C5:27  PH_B_FAULT_WRN_MIN %
% Rung: 9 %
SOR NEQ N11:0 N9:11 NEQ N11:0 N9:10 NEQ I:4.6 N7:88 BST GEQ I:4.6 N7:34 BST MOV N7:32 T4:10.PRE NXB XIC N7:1/6 TON T4:10 1.0 5 0 BND NXB GEQ I:4.6 N7:35 BST MOV N7:33 T4:11.PRE NXB XIC N7:3/6 TON T4:11 1.0 5 0 NXB XIC T4:11/DN OTE N17:7/7 BND BND EOR
%   N11:0  PROC_STATE  "STATE The current state of the process" %
%   N9:11  PROC_REGEN_B  "STATE Process Purify A" %
%   N9:10  PROCESS_STANDBY %
%   I:4.6  ADS_B_BED_TEMP  "Adsorber B TC8 bed temp C" %
%   N7:88  TC_OPEN_SP  "CONFIG The value read by an open TC input" %
%   N7:34  HT_PURIFY_ALM_SP  "CONFIG Purify High Temp Alarm Setpoint" %
%   N7:32  HT_PURIFY_ALM_DLY  "CONFIG Purify High Temp Alarm Delay" %
%   T4:10  PFY_HT_ADS_B_ALM_TMR  "TIMER Purify High Temp ADS B Alarm Delay" %
%   N7:1/6  HT_PURIFY_ALM_EN  "CONFIG Purify High Temp Alarm Enabled" %
%   N7:35  HT_PURIFY_WRN_SP  "CONFIG Purify High Temp Warning Setpoint" %
%   N7:33  HT_PURIFY_WRN_DLY  "CONFIG Purify High Temp Warning Delay" %
%   T4:11  PFY_HT_ADS_B_WRN_TMR  "TIMER Purify High Temp ADS B Warning Delay" %
%   N7:3/6  HT_PURIFY_WRN_EN  "CONFIG Purify High Temp Warning Enable" %
%   N17:7/7  HT_PURIFY_B_WARN  "WARNING ADS B Purify High Temp" %
% Rung: 10 %
SOR BST XIC T4:10/DN NXB XIC N17:5/7 XIO B31:4/0 XIO B31:2/0 BND OTE N17:5/7 EOR
%   T4:10  PFY_HT_ADS_B_ALM_TMR  "TIMER Purify High Temp ADS B Alarm Delay" %
%   N17:5/7  HT_PURIFY_B_ALARM  "ALARM ADS B Purify High Temp" %
%   B31:4/0  REGEN_RESUME  "COMMAND HMI Regen Resume" %
%   B31:2/0  START  "COMMAND HMI Start the process" %

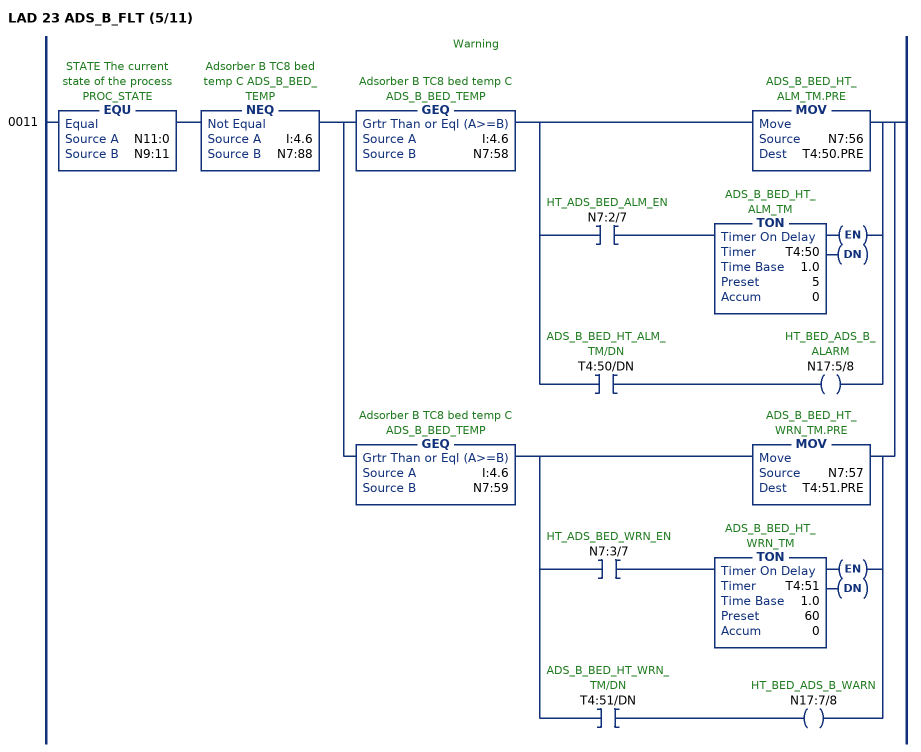
% Rung: 11 %
% Warning %
SOR EQU N11:0 N9:11 NEQ I:4.6 N7:88 BST GEQ I:4.6 N7:58 BST MOV N7:56 T4:50.PRE NXB XIC N7:2/7 TON T4:50 1.0 5 0 NXB XIC T4:50/DN OTE N17:5/8 BND NXB GEQ I:4.6 N7:59 BST MOV N7:57 T4:51.PRE NXB XIC N7:3/7 TON T4:51 1.0 60 0 NXB XIC T4:51/DN OTE N17:7/8 BND BND EOR
%   N11:0  PROC_STATE  "STATE The current state of the process" %
%   N9:11  PROC_REGEN_B  "STATE Process Purify A" %
%   I:4.6  ADS_B_BED_TEMP  "Adsorber B TC8 bed temp C" %
%   N7:88  TC_OPEN_SP  "CONFIG The value read by an open TC input" %
%   N7:58  HT_ADS_BED_ALM_SP %
%   N7:56  HT_ADS_BED_ALM_DLY %
%   T4:50  ADS_B_BED_HT_ALM_TM %
%   N7:2/7  HT_ADS_BED_ALM_EN %
%   N17:5/8  HT_BED_ADS_B_ALARM %
%   N7:59  HT_ADS_BED_WRN_SP %
%   N7:57  HT_ADS_BED_WRN_DLY %
%   T4:51  ADS_B_BED_HT_WRN_TM %
%   N7:3/7  HT_ADS_BED_WRN_EN %
%   N17:7/8  HT_BED_ADS_B_WARN %

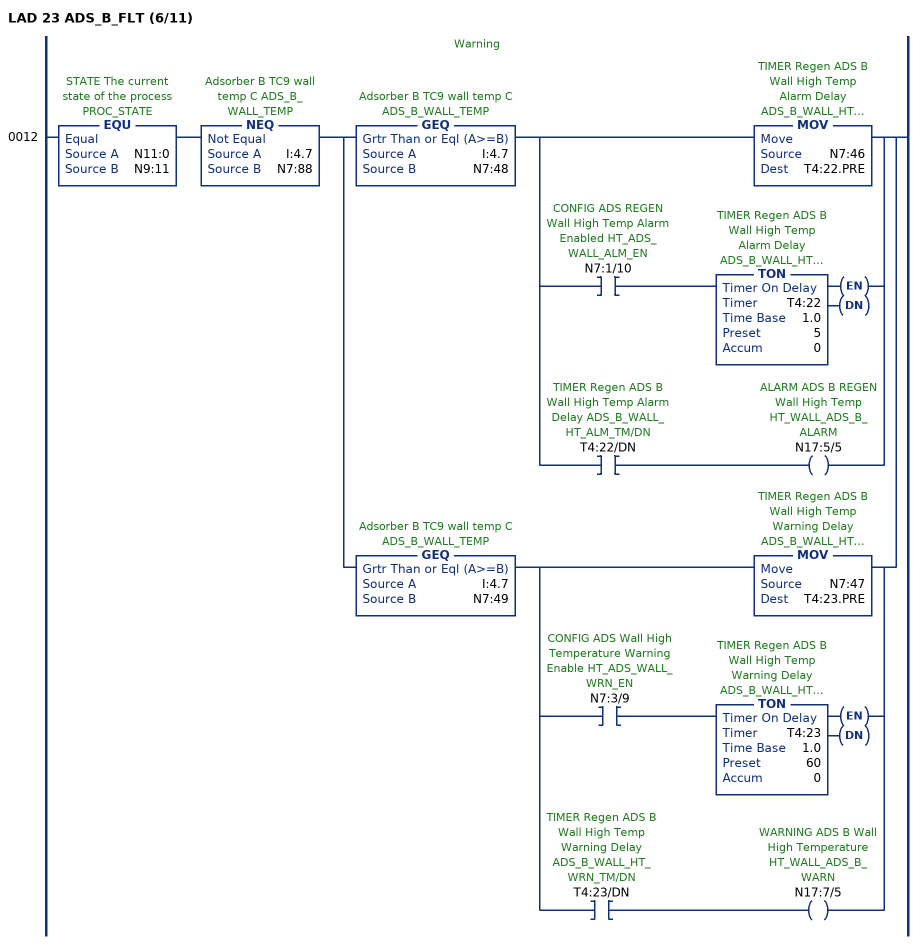
% Rung: 12 %
% Warning %
SOR EQU N11:0 N9:11 NEQ I:4.7 N7:88 BST GEQ I:4.7 N7:48 BST MOV N7:46 T4:22.PRE NXB XIC N7:1/10 TON T4:22 1.0 5 0 NXB XIC T4:22/DN OTE N17:5/5 BND NXB GEQ I:4.7 N7:49 BST MOV N7:47 T4:23.PRE NXB XIC N7:3/9 TON T4:23 1.0 60 0 NXB XIC T4:23/DN OTE N17:7/5 BND BND EOR
%   N11:0  PROC_STATE  "STATE The current state of the process" %
%   N9:11  PROC_REGEN_B  "STATE Process Purify A" %
%   I:4.7  ADS_B_WALL_TEMP  "Adsorber B TC9 wall temp C" %
%   N7:88  TC_OPEN_SP  "CONFIG The value read by an open TC input" %
%   N7:48  HT_ADS_WALL_ALM_SP  "CONFIG ADS Wall Regen High Temp Alarm" %
%   N7:46  HT_ADS_WALL_ALM_DLY  "CONFIG ADS Wall High Temperature Alarm Delay" %
%   T4:22  ADS_B_WALL_HT_ALM_TM  "TIMER Regen ADS B Wall High Temp Alarm Delay" %
%   N7:1/10  HT_ADS_WALL_ALM_EN  "CONFIG ADS REGEN Wall High Temp Alarm Enabled" %
%   N17:5/5  HT_WALL_ADS_B_ALARM  "ALARM ADS B REGEN Wall High Temp" %
%   N7:49  HT_ADS_WALL_WRN_SP  "CONFIG ADS Wall Regen High Temp Alarm" %
%   N7:47  HT_ADS_WALL_WRN_DLY  "CONFIG ADS Wall High Temperature Warning Delay" %
%   T4:23  ADS_B_WALL_HT_WRN_TM  "TIMER Regen ADS B Wall High Temp Warning Delay" %
%   N7:3/9  HT_ADS_WALL_WRN_EN  "CONFIG ADS Wall High Temperature Warning Enable" %
%   N17:7/5  HT_WALL_ADS_B_WARN  "WARNING ADS B Wall High Temperature" %

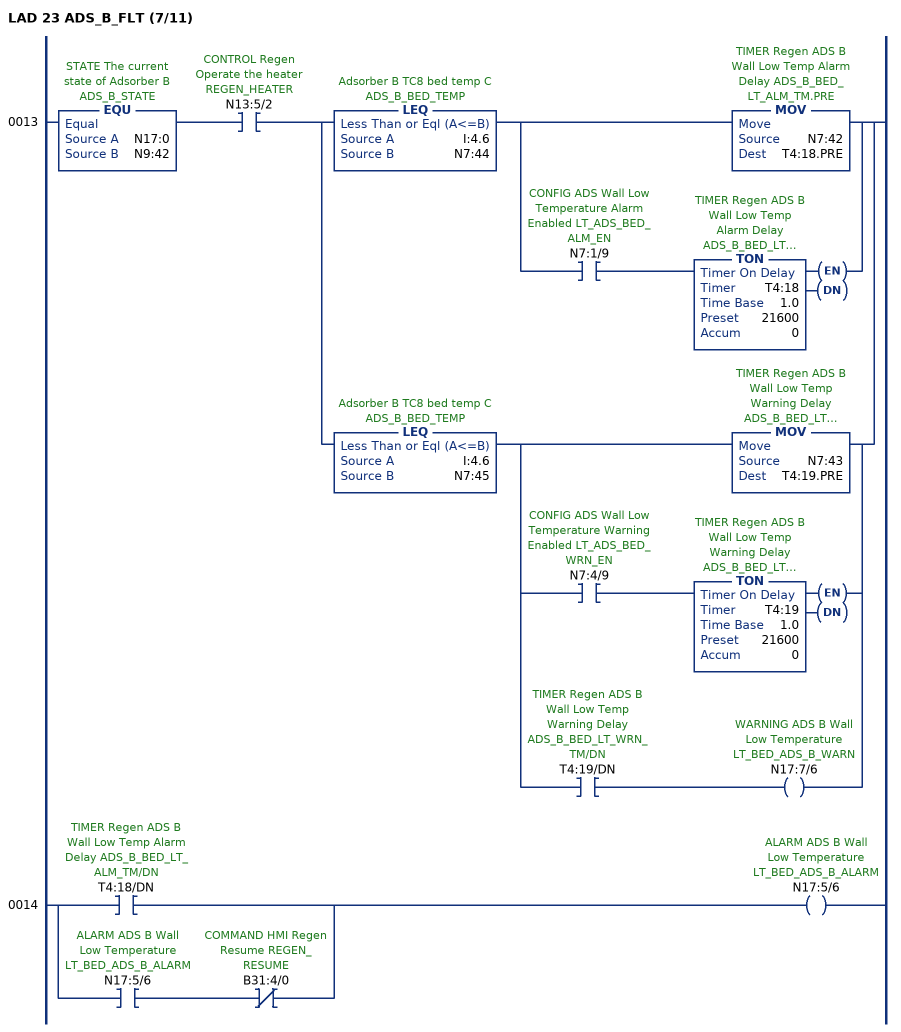
% Rung: 13 %
SOR EQU N17:0 N9:42 XIC N13:5/2 BST LEQ I:4.6 N7:44 BST MOV N7:42 T4:18.PRE NXB XIC N7:1/9 TON T4:18 1.0 21600 0 BND NXB LEQ I:4.6 N7:45 BST MOV N7:43 T4:19.PRE NXB XIC N7:4/9 TON T4:19 1.0 21600 0 NXB XIC T4:19/DN OTE N17:7/6 BND BND EOR
%   N17:0  ADS_B_STATE  "STATE The current state of Adsorber B" %
%   N9:42  ADS_REGEN  "STATE ADS Regen" %
%   N13:5/2  REGEN_HEATER  "CONTROL Regen Operate the heater" %
%   I:4.6  ADS_B_BED_TEMP  "Adsorber B TC8 bed temp C" %
%   N7:44  LT_ADS_BED_ALM_SP  "CONFIG ADS Wall Regen Heat Low Temperature Alarm Setpoint" %
%   N7:42  LT_ADS_BED_ALM_DLY  "CONFIG ADS Wall Regen heat Low Temperature Alarm Delay" %
%   T4:18  ADS_B_BED_LT_ALM_TM  "TIMER Regen ADS B Wall Low Temp Alarm Delay" %
%   N7:1/9  LT_ADS_BED_ALM_EN  "CONFIG ADS Wall Low Temperature Alarm Enabled" %
%   N7:45  LT_ADS_BED_WRN_SP  "CONFIG ADS Wall Regen Heat Low Temperature Warning Setpoint" %
%   N7:43  LT_ADS_BED_WRN_DLY  "CONFIG ADS Wall Regen heat Low Temperature Warning Delay" %
%   T4:19  ADS_B_BED_LT_WRN_TM  "TIMER Regen ADS B Wall Low Temp Warning Delay" %
%   N7:4/9  LT_ADS_BED_WRN_EN  "CONFIG ADS Wall Low Temperature Warning Enabled" %
%   N17:7/6  LT_BED_ADS_B_WARN  "WARNING ADS B Wall Low Temperature" %
% Rung: 14 %
SOR BST XIC T4:18/DN NXB XIC N17:5/6 XIO B31:4/0 BND OTE N17:5/6 EOR
%   T4:18  ADS_B_BED_LT_ALM_TM  "TIMER Regen ADS B Wall Low Temp Alarm Delay" %
%   N17:5/6  LT_BED_ADS_B_ALARM  "ALARM ADS B Wall Low Temperature" %
%   B31:4/0  REGEN_RESUME  "COMMAND HMI Regen Resume" %

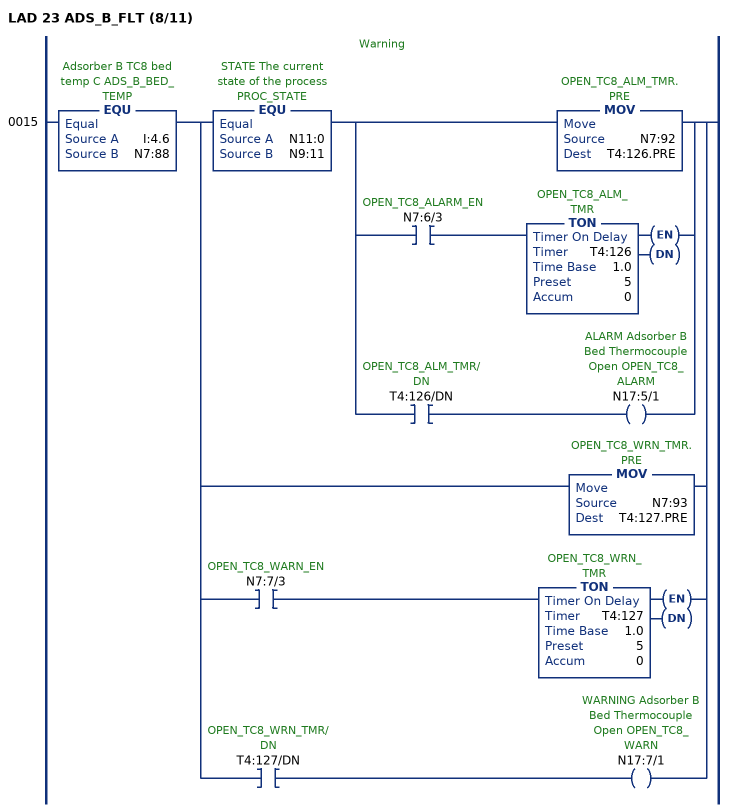
% Rung: 15 %
% Warning %
SOR EQU I:4.6 N7:88 BST EQU N11:0 N9:11 BST MOV N7:92 T4:126.PRE NXB XIC N7:6/3 TON T4:126 1.0 5 0 NXB XIC T4:126/DN OTE N17:5/1 BND NXB MOV N7:93 T4:127.PRE NXB XIC N7:7/3 TON T4:127 1.0 5 0 NXB XIC T4:127/DN OTE N17:7/1 BND EOR
%   I:4.6  ADS_B_BED_TEMP  "Adsorber B TC8 bed temp C" %
%   N7:88  TC_OPEN_SP  "CONFIG The value read by an open TC input" %
%   N11:0  PROC_STATE  "STATE The current state of the process" %
%   N9:11  PROC_REGEN_B  "STATE Process Purify A" %
%   N7:92  OPEN_TC_ALM_DLY %
%   T4:126  OPEN_TC8_ALM_TMR %
%   N7:6/3  OPEN_TC8_ALARM_EN %
%   N17:5/1  OPEN_TC8_ALARM  "ALARM Adsorber B Bed Thermocouple Open" %
%   N7:93  OPEN_TC_WRN_DLY %
%   T4:127  OPEN_TC8_WRN_TMR %
%   N7:7/3  OPEN_TC8_WARN_EN %
%   N17:7/1  OPEN_TC8_WARN  "WARNING Adsorber B Bed Thermocouple Open" %

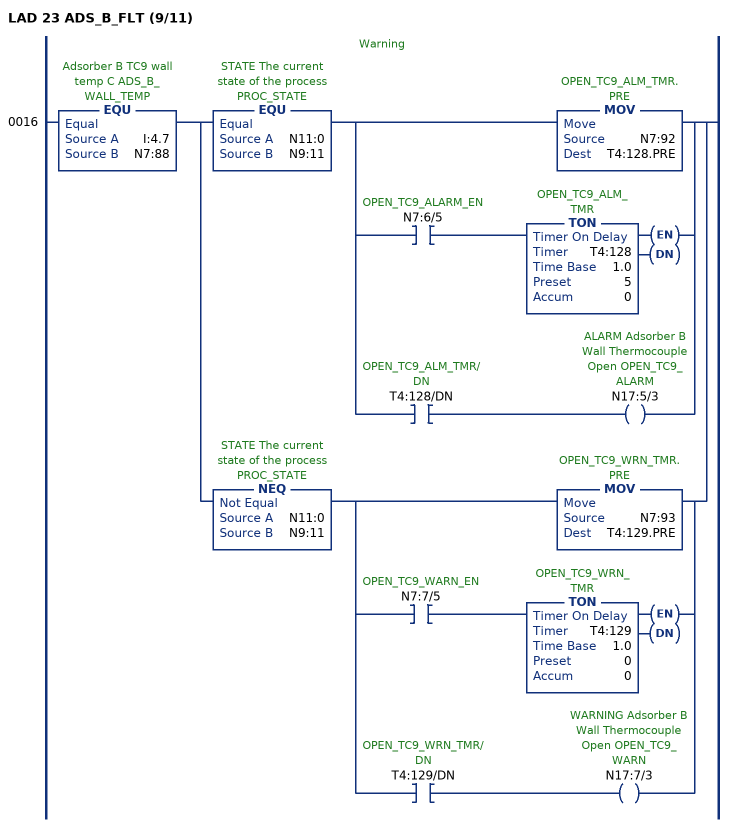
% Rung: 16 %
% Warning %
SOR EQU I:4.7 N7:88 BST EQU N11:0 N9:11 BST MOV N7:92 T4:128.PRE NXB XIC N7:6/5 TON T4:128 1.0 5 0 NXB XIC T4:128/DN OTE N17:5/3 BND NXB NEQ N11:0 N9:11 BST MOV N7:93 T4:129.PRE NXB XIC N7:7/5 TON T4:129 1.0 0 0 NXB XIC T4:129/DN OTE N17:7/3 BND BND EOR
%   I:4.7  ADS_B_WALL_TEMP  "Adsorber B TC9 wall temp C" %
%   N7:88  TC_OPEN_SP  "CONFIG The value read by an open TC input" %
%   N11:0  PROC_STATE  "STATE The current state of the process" %
%   N9:11  PROC_REGEN_B  "STATE Process Purify A" %
%   N7:92  OPEN_TC_ALM_DLY %
%   T4:128  OPEN_TC9_ALM_TMR %
%   N7:6/5  OPEN_TC9_ALARM_EN %
%   N17:5/3  OPEN_TC9_ALARM  "ALARM Adsorber B Wall Thermocouple Open" %
%   N7:93  OPEN_TC_WRN_DLY %
%   T4:129  OPEN_TC9_WRN_TMR %
%   N7:7/5  OPEN_TC9_WARN_EN %
%   N17:7/3  OPEN_TC9_WARN  "WARNING Adsorber B Wall Thermocouple Open" %

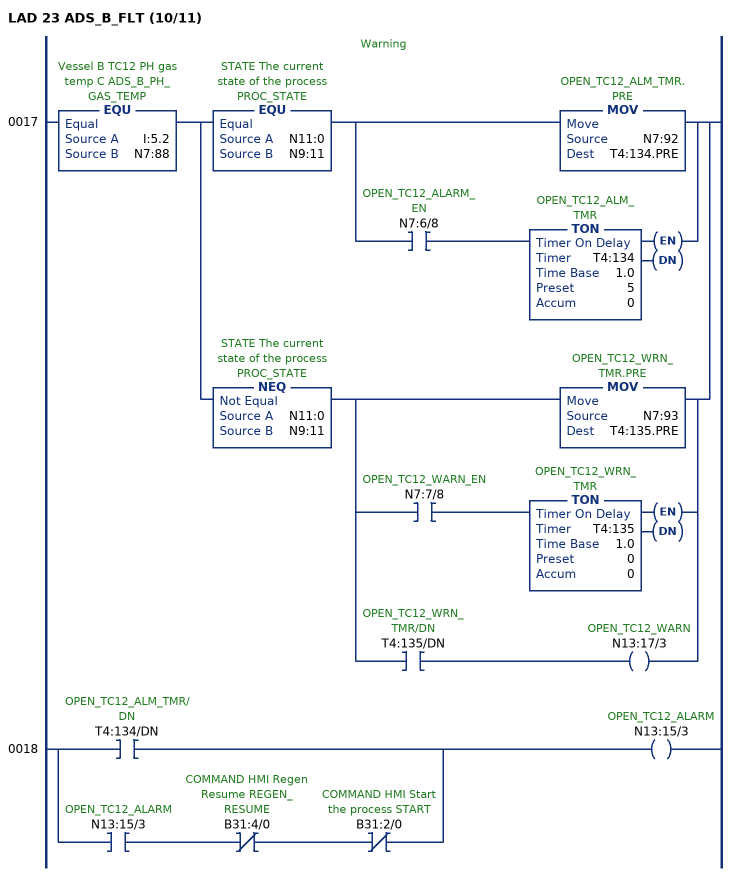
% Rung: 17 %
% Warning %
SOR EQU I:5.2 N7:88 BST EQU N11:0 N9:11 BST MOV N7:92 T4:134.PRE NXB XIC N7:6/8 TON T4:134 1.0 5 0 BND NXB NEQ N11:0 N9:11 BST MOV N7:93 T4:135.PRE NXB XIC N7:7/8 TON T4:135 1.0 0 0 NXB XIC T4:135/DN OTE N13:17/3 BND BND EOR
%   I:5.2  ADS_B_PH_GAS_TEMP  "Vessel B TC12 PH gas temp C" %
%   N7:88  TC_OPEN_SP  "CONFIG The value read by an open TC input" %
%   N11:0  PROC_STATE  "STATE The current state of the process" %
%   N9:11  PROC_REGEN_B  "STATE Process Purify A" %
%   N7:92  OPEN_TC_ALM_DLY %
%   T4:134  OPEN_TC12_ALM_TMR %
%   N7:6/8  OPEN_TC12_ALARM_EN %
%   N7:93  OPEN_TC_WRN_DLY %
%   T4:135  OPEN_TC12_WRN_TMR %
%   N7:7/8  OPEN_TC12_WARN_EN %
%   N13:17/3  OPEN_TC12_WARN %
% Rung: 18 %
SOR BST XIC T4:134/DN NXB XIC N13:15/3 XIO B31:4/0 XIO B31:2/0 BND OTE N13:15/3 EOR
%   T4:134  OPEN_TC12_ALM_TMR %
%   N13:15/3  OPEN_TC12_ALARM %
%   B31:4/0  REGEN_RESUME  "COMMAND HMI Regen Resume" %
%   B31:2/0  START  "COMMAND HMI Start the process" %

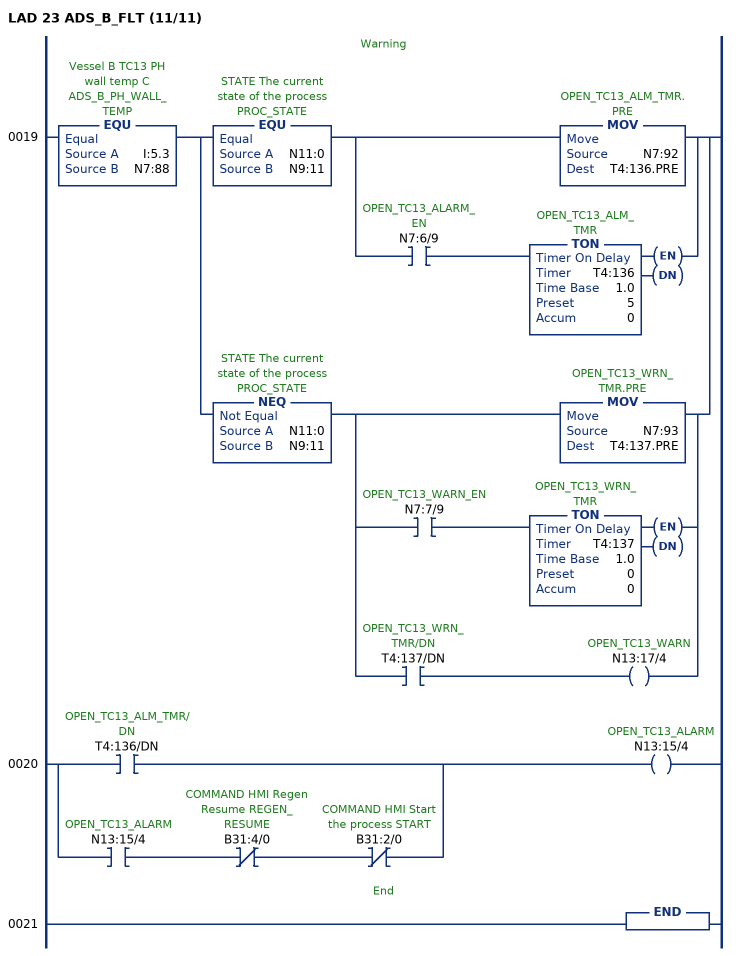
% Rung: 19 %
% Warning %
SOR EQU I:5.3 N7:88 BST EQU N11:0 N9:11 BST MOV N7:92 T4:136.PRE NXB XIC N7:6/9 TON T4:136 1.0 5 0 BND NXB NEQ N11:0 N9:11 BST MOV N7:93 T4:137.PRE NXB XIC N7:7/9 TON T4:137 1.0 0 0 NXB XIC T4:137/DN OTE N13:17/4 BND BND EOR
%   I:5.3  ADS_B_PH_WALL_TEMP  "Vessel B TC13 PH wall temp C" %
%   N7:88  TC_OPEN_SP  "CONFIG The value read by an open TC input" %
%   N11:0  PROC_STATE  "STATE The current state of the process" %
%   N9:11  PROC_REGEN_B  "STATE Process Purify A" %
%   N7:92  OPEN_TC_ALM_DLY %
%   T4:136  OPEN_TC13_ALM_TMR %
%   N7:6/9  OPEN_TC13_ALARM_EN %
%   N7:93  OPEN_TC_WRN_DLY %
%   T4:137  OPEN_TC13_WRN_TMR %
%   N7:7/9  OPEN_TC13_WARN_EN %
%   N13:17/4  OPEN_TC13_WARN %
% Rung: 20 %
SOR BST XIC T4:136/DN NXB XIC N13:15/4 XIO B31:4/0 XIO B31:2/0 BND OTE N13:15/4 EOR
%   T4:136  OPEN_TC13_ALM_TMR %
%   N13:15/4  OPEN_TC13_ALARM %
%   B31:4/0  REGEN_RESUME  "COMMAND HMI Regen Resume" %
%   B31:2/0  START  "COMMAND HMI Start the process" %
% Rung: 21 %
% End %
SOR END EOR

LADDER 49 "MODBUS"
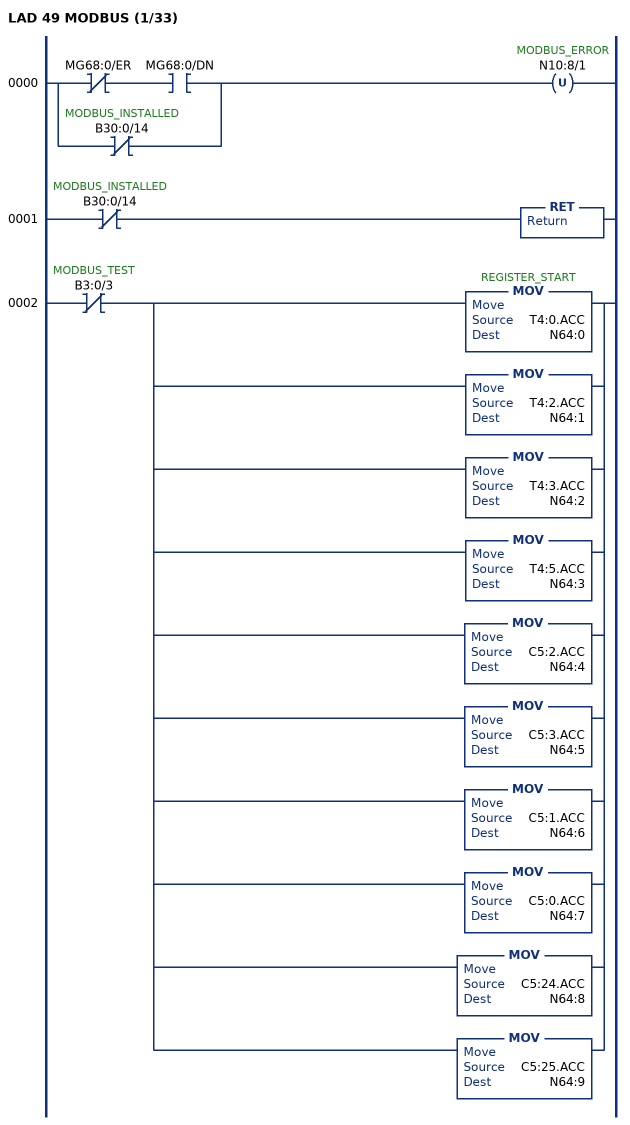
% Rung: 0 %
SOR BST XIO MG68:0/ER XIC MG68:0/DN NXB XIO B30:0/14 BND OTU N10:8/1 EOR
%   B30:0/14  MODBUS_INSTALLED %
%   N10:8/1  MODBUS_ERROR %
% Rung: 1 %
SOR XIO B30:0/14 RET EOR
%   B30:0/14  MODBUS_INSTALLED %
% Rung: 2 %
SOR XIO B3:0/3 BST MOV T4:0.ACC N64:0 NXB MOV T4:2.ACC N64:1 NXB MOV T4:3.ACC N64:2 NXB MOV T4:5.ACC N64:3 NXB MOV C5:2.ACC N64:4 NXB MOV C5:3.ACC N64:5 NXB MOV C5:1.ACC N64:6 NXB MOV C5:0.ACC N64:7 NXB MOV C5:24.ACC N64:8 NXB MOV C5:25.ACC N64:9 BND EOR
%   B3:0/3  MODBUS_TEST %
%   T4:0  PURIFY_OVERLAP_SEC  "TIMER Purify Overlap" %
%   N64:0  REGISTER_START %
%   T4:2  REGEN_DELAY_TIMER  "TIMER Regen Delay (seconds)" %
%   T4:3  REGEN_VENT_SEC_TMR  "TIMER Regen Vent (seconds)" %
%   T4:5  REGEN_COOL_SEC_TIMER  "TIMER Regen Cool (seconds)" %
%   C5:2  PURIFY_ACTIVE_TTL_HR  "COUNTER The number of total elapsed purification hours for the process equipment" %
%   C5:3  PURIFY_ACTIVE_TTL_DY  "COUNTER The number of total elapsed purification days for the process equipment" %
%   C5:1  PURIFY_ACTIVE_MINUTE  "COUNTER The number of elapsed purification minutes for the current ADS (60 min)" %
%   C5:0  PURIFY_ACTIVE_HOURS  "COUNTER The number of elapsed purification hours for the current ADS" %
%   C5:24  REGEN_VENT_MIN_CTR %
%   C5:25  REGEN_VENT_HRS_CTR %

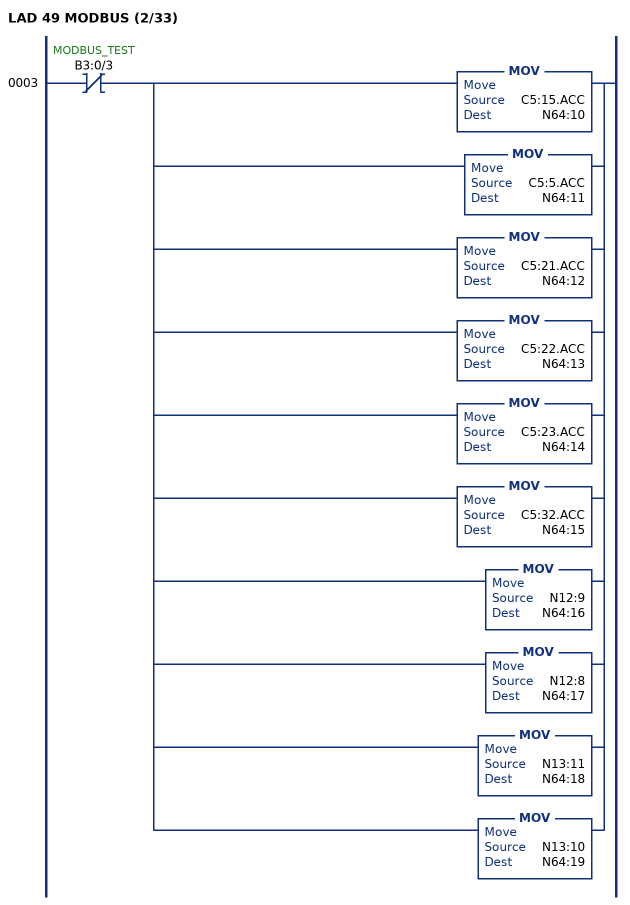
% Rung: 3 %
SOR XIO B3:0/3 BST MOV C5:15.ACC N64:10 NXB MOV C5:5.ACC N64:11 NXB MOV C5:21.ACC N64:12 NXB MOV C5:22.ACC N64:13 NXB MOV C5:23.ACC N64:14 NXB MOV C5:32.ACC N64:15 NXB MOV N12:9 N64:16 NXB MOV N12:8 N64:17 NXB MOV N13:11 N64:18 NXB MOV N13:10 N64:19 BND EOR
%   B3:0/3  MODBUS_TEST %
%   C5:15  REGEN_RUN_MINUTE %
%   C5:5  REGEN_COOL_MINUTE  "COUNTER Regen the number of minutes for which the bed has cooled" %
%   C5:21  REGEN_EQUALIZE_MIN %
%   C5:22  REGEN_COND_MIN_CTR %
%   C5:23  REGEN_COND_HRS_CTR %
%   C5:32  PURIFY_OVERLAP_MIN %
%   N12:9  MIN_LEFT_IN_PURIFY %
%   N12:8  HRS_LEFT_IN_PURIFY %
%   N13:11  REGEN_MIN_LEFT %
%   N13:10  REGEN_HRS_LEFT %

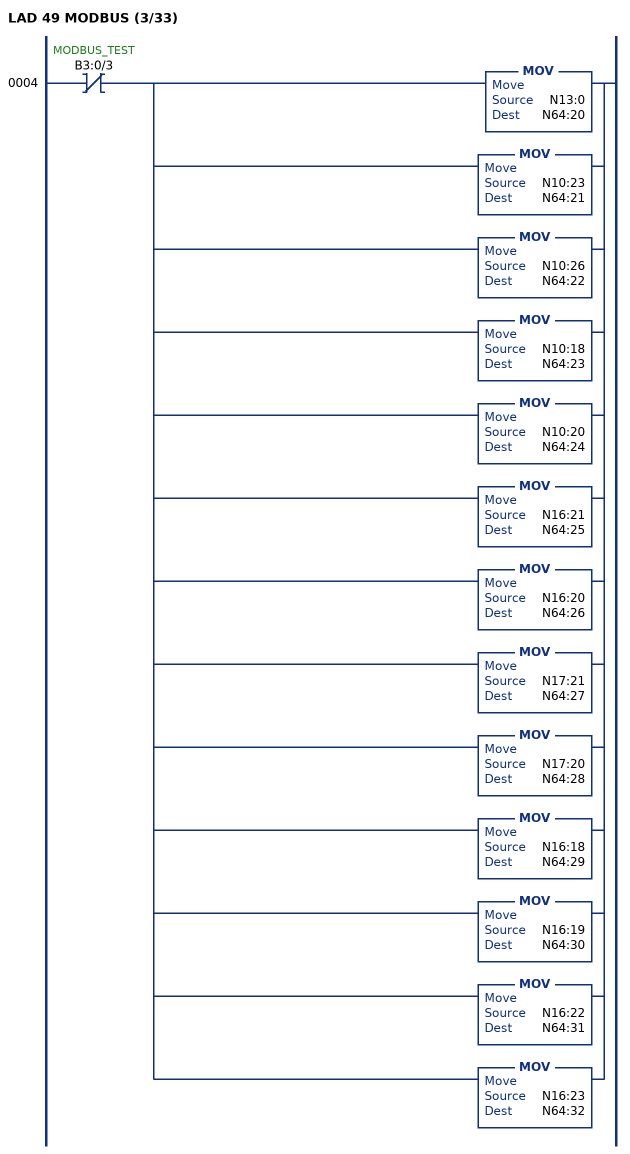
% Rung: 4 %
SOR XIO B3:0/3 BST MOV N13:0 N64:20 NXB MOV N10:23 N64:21 NXB MOV N10:26 N64:22 NXB MOV N10:18 N64:23 NXB MOV N10:20 N64:24 NXB MOV N16:21 N64:25 NXB MOV N16:20 N64:26 NXB MOV N17:21 N64:27 NXB MOV N17:20 N64:28 NXB MOV N16:18 N64:29 NXB MOV N16:19 N64:30 NXB MOV N16:22 N64:31 NXB MOV N16:23 N64:32 BND EOR
%   B3:0/3  MODBUS_TEST %
%   N13:0  REGEN_STATE  "<datalog> The current state of the regen process" %
%   N10:23  MOISTURE_SENSOR_TEMP  "<datalog> Moisture sensor MS-1 temp C." %
%   N10:26  MFM_FLOW %
%   N10:18  INLET_PX_PSIG  "<datalog> Inlet pressure PX_1 in PSIG." %
%   N10:20  OUTLET_PX_PSIG  "<datalog> Outlet pressure PX-2 in PSIG." %
%   N16:21  ADS_A_BED_TEMP_READ  "<datalog> Adsorber A bed TC6 bed temp C" %
%   N16:20  ADS_A_WALL_TEMP_READ  "<datalog> Adsorber A wall TC7 bed temp C" %
%   N17:21  ADS_B_BED_TEMP_READ  "<datalog> Adsorber B bed TC8 bed temp C" %
%   N17:20  ADS_B_WALL_TEMP_READ  "<datalog> Adsorber B bed TC9 wall temp C" %
%   N16:18  PH_A_GAS_TEMP_READ  "<datalog> Adsorber A TC10 PH gas temp C" %
%   N16:19  PH_A_ROD_TEMP_READ  "<datalog>" %
%   N16:22  PH_B_GAS_TEMP_READ  "<datalog> Adsorber B TC12 PH gas temp C" %
%   N16:23  PH_B_ROD_TEMP_READ  "<datalog> Adsorber B TC13 PH wall temp C" %

